KUKA KRL program: MyProgram_272().src

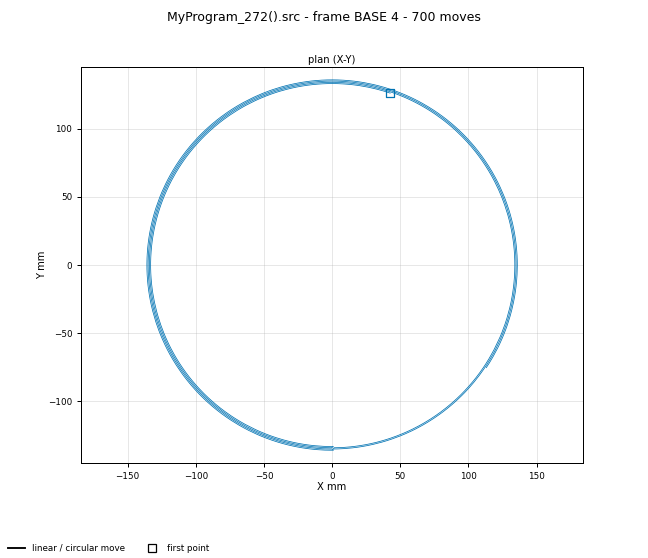
[picture p0: tool path of MyProgram_272().src in frame BASE 4, 700 of 700 moves have a stored position in this frame; points joined in program order, loops and branches not executed]
&ACCESS RVP
&REL 1
&PARAM TEMPLATE = C:\KRC\Roboter\Template\vorgabe
&PARAM EDITMASK = *
DEF MyProgram_272()
; ---- Setting reference (Base) ----
$BASE = BASE_DATA[4]

; --------------------------
; ---- Setting tool (TCP) ----
$TOOL = TOOL_DATA[3]
; --------------------------

$VEL.CP = VEL_APROX_PRINT
Startdeposition()
$VEL.CP = VEL_PRINT
LIN {X 42.5877,Y 126.1093,Z 171,A 71.929,B 9.2789,C 0.0558,E1 9.3306,E2 379.3226} C_DIS
LIN {X 38.192,Y 127.5107,Z 171,A 74.1551,B 9.2789,C 0.0493,E1 9.3246,E2 377.0683} C_DIS
LIN {X 32.5615,Y 129.0611,Z 171,A 76.4995,B 9.2789,C 0.0509,E1 9.3183,E2 374.7445} C_DIS
LIN {X 29.5199,Y 129.7905,Z 171,A 77.8234,B 9.2789,C 0.0505,E1 9.3147,E2 373.4236} C_DIS
LIN {X 26.303,Y 130.4807,Z 171,A 79.258,B 9.2789,C 0.0493,E1 9.3108,E2 371.9872} C_DIS
LIN {X 23.1123,Y 131.0837,Z 171,A 80.6058,B 9.2789,C 0.0496,E1 9.3071,E2 370.6457} C_DIS
LIN {X 20.0394,Y 131.5886,Z 171,A 81.9788,B 9.2789,C 0.0484,E1 9.3033,E2 369.2693} C_DIS
LIN {X 16.1157,Y 132.1266,Z 171,A 83.746,B 9.2789,C 0.0466,E1 9.2984,E2 367.4952} C_DIS
LIN {X 12.5078,Y 132.5166,Z 171,A 85.3108,B 9.2789,C 0.0461,E1 9.2941,E2 365.9307} C_DIS
LIN {X 8.3924,Y 132.8408,Z 171,A 87.0897,B 9.2789,C 0.0458,E1 9.2891,E2 364.1522} C_DIS
LIN {X 4.1202,Y 133.0424,Z 171,A 88.9439,B 9.2789,C 0.0454,E1 9.2839,E2 362.2973} C_DIS
LIN {X 0.5227,Y 133.1047,Z 171,A 90.4815,B 9.2789,C 0.0456,E1 9.2796,E2 360.7616} C_DIS
LIN {X -3.6809,Y 133.0546,Z 171,A 92.2437,B 9.2789,C 0.0466,E1 9.2747,E2 359.006} C_DIS
LIN {X -7.0154,Y 132.9209,Z 171,A 93.6521,B 9.2789,C 0.0474,E1 9.2708,E2 357.6017} C_DIS
LIN {X -10.707,Y 132.675,Z 171,A 95.3254,B 9.2789,C 0.0462,E1 9.2661,E2 355.9196} C_DIS
LIN {X -14.2828,Y 132.3368,Z 171,A 96.8212,B 9.2789,C 0.0477,E1 9.262,E2 354.4306} C_DIS
LIN {X -17.8991,Y 131.8978,Z 171,A 98.5277,B 9.2789,C 0.0457,E1 9.2572,E2 352.7086} C_DIS
LIN {X -21.9542,Y 131.2822,Z 171,A 100.1748,B 9.2789,C 0.0488,E1 9.2527,E2 351.0765} C_DIS
LIN {X -25.7118,Y 130.6003,Z 171,A 101.7895,B 9.2789,C 0.0503,E1 9.2483,E2 349.4665} C_DIS
LIN {X -29.321,Y 129.836,Z 171,A 103.4986,B 9.2789,C 0.049,E1 9.2436,E2 347.7439} C_DIS
LIN {X -33.1581,Y 128.9097,Z 171,A 105.1133,B 9.2789,C 0.0518,E1 9.2393,E2 346.1403} C_DIS
LIN {X -38.1705,Y 127.5171,Z 171,A 107.3466,B 9.2789,C 0.0538,E1 9.2333,E2 343.9094} C_DIS
LIN {X -40.8644,Y 126.6776,Z 171,A 108.5976,B 9.2789,C 0.0542,E1 9.2299,E2 342.6549} C_DIS
LIN {X -44.5339,Y 125.4356,Z 171,A 110.3593,B 9.2789,C 0.0542,E1 9.2253,E2 340.8833} C_DIS
LIN {X -48.093,Y 124.1129,Z 171,A 112.4224,B 9.2789,C 0.0481,E1 9.2198,E2 338.7703} C_DIS
LIN {X -52.2312,Y 122.4306,Z 171,A 113.7596,B 9.2789,C 0.0609,E1 9.2165,E2 337.5044} C_DIS
LIN {X -56.3646,Y 120.583,Z 171,A 115.8018,B 9.2789,C 0.0616,E1 9.2113,E2 335.4528} C_DIS
LIN {X -60.1833,Y 118.7221,Z 171,A 117.4022,B 9.2789,C 0.0681,E1 9.2073,E2 333.8809} C_DIS
LIN {X -62.74,Y 117.3935,Z 171,A 118.8099,B 9.2789,C 0.0669,E1 9.2038,E2 332.4544} C_DIS
LIN {X -65.4527,Y 115.9029,Z 171,A 120.3033,B 9.2789,C 0.0659,E1 9.2001,E2 330.9431} C_DIS
LIN {X -69.1961,Y 113.7079,Z 171,A 122.2249,B 9.2789,C 0.0678,E1 9.1955,E2 329.0167} C_DIS
LIN {X -73.1227,Y 111.2229,Z 171,A 123.9787,B 9.2788,C 0.0753,E1 9.1915,E2 327.2939} C_DIS
LIN {X -75.3901,Y 109.6986,Z 171,A 126.0091,B 9.2788,C 0.0623,E1 9.1866,E2 325.1627} C_DIS
LIN {X -79.6378,Y 106.655,Z 171,A 128.1469,B 9.2788,C 0.0683,E1 9.1818,E2 323.0405} C_DIS
LIN {X -83.2399,Y 103.8687,Z 171,A 129.6575,B 9.2788,C 0.0797,E1 9.1786,E2 321.5854} C_DIS
LIN {X -86.59,Y 101.0928,Z 171,A 131.612,B 9.2788,C 0.0818,E1 9.1744,E2 319.623} C_DIS
LIN {X -90.0311,Y 98.0401,Z 171,A 133.5166,B 9.2787,C 0.087,E1 9.1705,E2 317.7292} C_DIS
LIN {X -93.0134,Y 95.2157,Z 171,A 135.3296,B 9.2787,C 0.0899,E1 9.1669,E2 315.9127} C_DIS
LIN {X -95.7889,Y 92.4229,Z 171,A 137.1312,B 9.2787,C 0.0916,E1 9.1633,E2 314.1} C_DIS
LIN {X -99.0111,Y 88.9624,Z 171,A 139.1371,B 9.2786,C 0.0966,E1 9.1595,E2 312.0998} C_DIS
LIN {X -101.9431,Y 85.5866,Z 171,A 141.0403,B 9.2786,C 0.1012,E1 9.1561,E2 310.201} C_DIS
LIN {X -104.4924,Y 82.4553,Z 171,A 142.8577,B 9.2785,C 0.1039,E1 9.1529,E2 308.376} C_DIS
LIN {X -107.2539,Y 78.8293,Z 171,A 145.3979,B 9.2785,C 0.0988,E1 9.1486,E2 305.7684} C_DIS
LIN {X -110.2026,Y 74.6515,Z 171,A 147.0279,B 9.2784,C 0.1137,E1 9.1461,E2 304.2093} C_DIS
LIN {X -112.3849,Y 71.3246,Z 171,A 148.7665,B 9.2784,C 0.1175,E1 9.1435,E2 302.4694} C_DIS
LIN {X -114.8083,Y 67.3536,Z 171,A 150.9264,B 9.2784,C 0.1199,E1 9.1404,E2 300.2927} C_DIS
LIN {X -117.651,Y 62.2522,Z 171,A 153.1134,B 9.2781,C 0.1318,E1 9.1375,E2 298.1473} C_DIS
LIN {X -119.7398,Y 58.1376,Z 171,A 155.2917,B 9.2781,C 0.1338,E1 9.1347,E2 295.9483} C_DIS
LIN {X -121.0064,Y 55.4489,Z 171,A 156.578,B 9.2781,C 0.1371,E1 9.1332,E2 294.6624} C_DIS
LIN {X -122.3225,Y 52.4813,Z 171,A 158.0107,B 9.2781,C 0.1403,E1 9.1316,E2 293.227} C_DIS
LIN {X -123.8951,Y 48.6534,Z 171,A 159.9678,B 9.278,C 0.1422,E1 9.1296,E2 291.2507} C_DIS
LIN {X -125.2945,Y 44.9253,Z 171,A 161.607,B 9.278,C 0.1482,E1 9.128,E2 289.6223} C_DIS
LIN {X -126.5325,Y 41.3167,Z 171,A 163.3756,B 9.2779,C 0.1507,E1 9.1264,E2 287.8403} C_DIS
LIN {X -127.7786,Y 37.2777,Z 171,A 165.1311,B 9.2778,C 0.1568,E1 9.125,E2 286.0943} C_DIS
LIN {X -128.6977,Y 33.9703,Z 171,A 166.6461,B 9.2778,C 0.1604,E1 9.1239,E2 284.5764} C_DIS
LIN {X -129.8767,Y 29.1424,Z 171,A 168.7116,B 9.2776,C 0.1677,E1 9.1226,E2 282.5219} C_DIS
LIN {X -130.5951,Y 25.7359,Z 171,A 170.9382,B 9.2777,C 0.16,E1 9.1214,E2 280.2091} C_DIS
LIN {X -131.4748,Y 20.7743,Z 171,A 172.311,B 9.2774,C 0.1793,E1 9.1208,E2 278.9345} C_DIS
LIN {X -131.9531,Y 17.4769,Z 171,A 173.9819,B 9.2774,C 0.1796,E1 9.1201,E2 277.2366} C_DIS
LIN {X -132.405,Y 13.649,Z 171,A 175.7439,B 9.2773,C 0.1827,E1 9.1196,E2 275.4639} C_DIS
LIN {X -132.7511,Y 9.7054,Z 171,A 177.3737,B 9.2772,C 0.1889,E1 9.1192,E2 273.8447} C_DIS
LIN {X -132.9834,Y 5.7253,Z 171,A 179.185,B 9.2772,C 0.1923,E1 9.119,E2 272.0236} C_DIS
LIN {X -133.0886,Y 2.1253,Z 171,A -179.3539,B 9.277,C 0.1983,E1 9.1189,E2 270.5747} C_DIS
LIN {X -133.089,Y -2.0987,Z 171,A -177.4486,B 9.2769,C 0.2021,E1 9.1189,E2 268.6607} C_DIS
LIN {X -132.9791,Y -5.8335,Z 171,A -175.7236,B 9.2769,C 0.2049,E1 9.1191,E2 266.9232} C_DIS
LIN {X -132.7452,Y -9.7862,Z 171,A -174.0656,B 9.2767,C 0.2106,E1 9.1194,E2 265.2722} C_DIS
LIN {X -132.3555,Y -14.1094,Z 171,A -172.1851,B 9.2766,C 0.2158,E1 9.1199,E2 263.392} C_DIS
LIN {X -131.8984,Y -17.8939,Z 171,A -170.5736,B 9.2765,C 0.221,E1 9.1205,E2 261.7855} C_DIS
LIN {X -131.3884,Y -21.3181,Z 171,A -168.1542,B 9.2767,C 0.2099,E1 9.1217,E2 259.2544} C_DIS
LIN {X -130.2557,Y -27.4034,Z 171,A -166.3772,B 9.2762,C 0.2321,E1 9.1226,E2 257.5877} C_DIS
LIN {X -128.6414,Y -34.1817,Z 171,A -162.9035,B 9.2762,C 0.2327,E1 9.1249,E2 254.0589} C_DIS
LIN {X -127.6689,Y -37.652,Z 171,A -161.671,B 9.2759,C 0.2423,E1 9.1259,E2 252.8664} C_DIS
LIN {X -126.5371,Y -41.303,Z 171,A -160.0341,B 9.2759,C 0.2469,E1 9.1272,E2 251.2318} C_DIS
LIN {X -125.5991,Y -44.0688,Z 171,A -158.7983,B 9.2757,C 0.2507,E1 9.1284,E2 249.9995} C_DIS
LIN {X -124.5345,Y -46.9914,Z 171,A -157.3661,B 9.2757,C 0.2527,E1 9.1298,E2 248.557} C_DIS
LIN {X -123.3937,Y -49.9094,Z 171,A -155.9581,B 9.2756,C 0.2553,E1 9.1312,E2 247.1427} C_DIS
LIN {X -122.0333,Y -53.15,Z 171,A -154.4655,B 9.2755,C 0.2597,E1 9.1329,E2 245.6536} C_DIS
LIN {X -119.9685,Y -57.6591,Z 171,A -152.3072,B 9.2753,C 0.2648,E1 9.1354,E2 243.4938} C_DIS
LIN {X -118.1397,Y -61.3214,Z 171,A -150.483,B 9.2753,C 0.2682,E1 9.1377,E2 241.6632} C_DIS
LIN {X -115.8549,Y -65.5381,Z 171,A -148.4796,B 9.2751,C 0.2744,E1 9.1404,E2 239.6686} C_DIS
LIN {X -113.9926,Y -68.7254,Z 171,A -146.718,B 9.2751,C 0.2754,E1 9.143,E2 237.8869} C_DIS
LIN {X -111.7318,Y -72.3428,Z 171,A -144.854,B 9.2749,C 0.2793,E1 9.1458,E2 236.0204} C_DIS
LIN {X -109.9906,Y -74.9641,Z 171,A -143.532,B 9.2748,C 0.2831,E1 9.1478,E2 234.7031} C_DIS
LIN {X -107.4993,Y -78.4952,Z 171,A -141.6558,B 9.2747,C 0.2871,E1 9.1509,E2 232.8259} C_DIS
LIN {X -104.9019,Y -81.9339,Z 171,A -139.7691,B 9.2746,C 0.2907,E1 9.1541,E2 230.9362} C_DIS
LIN {X -102.8056,Y -84.5496,Z 171,A -138.2669,B 9.2745,C 0.2928,E1 9.1568,E2 229.4274} C_DIS
LIN {X -99.9648,Y -87.8898,Z 171,A -136.4848,B 9.2743,C 0.2987,E1 9.16,E2 227.6589} C_DIS
LIN {X -97.5072,Y -90.608,Z 171,A -134.6846,B 9.2743,C 0.298,E1 9.1634,E2 225.8321} C_DIS
LIN {X -94.0902,Y -94.1522,Z 171,A -132.586,B 9.2742,C 0.3026,E1 9.1676,E2 223.7367} C_DIS
LIN {X -90.8102,Y -97.3189,Z 171,A -130.6365,B 9.2741,C 0.3066,E1 9.1715,E2 221.7895} C_DIS
LIN {X -87.8913,Y -99.9635,Z 171,A -128.9777,B 9.2739,C 0.3104,E1 9.1749,E2 220.1357} C_DIS
LIN {X -84.6172,Y -102.7497,Z 171,A -127.0049,B 9.2739,C 0.3115,E1 9.1792,E2 218.1483} C_DIS
LIN {X -81.9414,Y -104.8961,Z 171,A -125.5632,B 9.2738,C 0.3147,E1 9.1824,E2 216.7112} C_DIS
LIN {X -78.4506,Y -107.5319,Z 171,A -123.6313,B 9.2738,C 0.3169,E1 9.1867,E2 214.7736} C_DIS
LIN {X -73.7879,Y -110.7828,Z 171,A -121.4632,B 9.2734,C 0.3257,E1 9.1916,E2 212.6402} C_DIS
LIN {X -71.2924,Y -112.4052,Z 171,A -119.8915,B 9.2735,C 0.3223,E1 9.1954,E2 211.0329} C_DIS
LIN {X -67.4694,Y -114.7403,Z 171,A -117.9853,B 9.2735,C 0.3254,E1 9.2,E2 209.1296} C_DIS
LIN {X -63.5644,Y -116.949,Z 171,A -115.9592,B 9.2734,C 0.3262,E1 9.2049,E2 207.0919} C_DIS
LIN {X -56.1378,Y -120.6878,Z 171,A -112.7264,B 9.273,C 0.3369,E1 9.2129,E2 203.9018} C_DIS
LIN {X -52.728,Y -122.2158,Z 171,A -110.8624,B 9.2731,C 0.3338,E1 9.2178,E2 202.0062} C_DIS
LIN {X -48.8795,Y -123.8072,Z 171,A -109.1519,B 9.2731,C 0.3371,E1 9.2222,E2 200.3059} C_DIS
LIN {X -45.6244,Y -125.0425,Z 171,A -107.7189,B 9.2729,C 0.3397,E1 9.2259,E2 198.8808} C_DIS
LIN {X -41.1313,Y -126.5923,Z 171,A -105.3843,B 9.273,C 0.3359,E1 9.2322,E2 196.5103} C_DIS
LIN {X -35.3399,Y -128.329,Z 171,A -102.9247,B 9.2729,C 0.3405,E1 9.2387,E2 194.0678} C_DIS
LIN {X -31.3297,Y -129.3656,Z 171,A -101.1229,B 9.2729,C 0.3411,E1 9.2436,E2 192.2633} C_DIS
LIN {X -28.0532,Y -130.1154,Z 171,A -99.6907,B 9.2729,C 0.3422,E1 9.2475,E2 190.8326} C_DIS
LIN {X -24.622,Y -130.8087,Z 171,A -98.045,B 9.2729,C 0.3401,E1 9.2521,E2 189.1693} C_DIS
LIN {X -20.5153,Y -131.5149,Z 171,A -96.3614,B 9.2728,C 0.3429,E1 9.2567,E2 187.4987} C_DIS
LIN {X -16.8361,Y -132.0371,Z 171,A -94.6911,B 9.2728,C 0.3419,E1 9.2613,E2 185.8191} C_DIS
LIN {X -12.5397,Y -132.5135,Z 171,A -92.9033,B 9.2728,C 0.3437,E1 9.2663,E2 184.0396} C_DIS
LIN {X -9.3135,Y -132.7797,Z 171,A -91.5471,B 9.2728,C 0.3446,E1 9.27,E2 182.6876} C_DIS
LIN {X -6.5086,Y -132.9463,Z 171,A -90.3022,B 9.2728,C 0.3439,E1 9.2735,E2 181.4378} C_DIS
LIN {X -2.5391,Y -133.0817,Z 171,A -88.4788,B 9.2728,C 0.3415,E1 9.2786,E2 179.5995} C_DIS
LIN {X 0.9624,Y -133.1014,Z 171,A -87.5259,B 9.2724,C 0.3524,E1 9.2811,E2 178.7143} C_DIS
Enddeposition()
LIN {X 0.9624,Y -133.1014,Z 171,A -87.5259,B 9.2724,C 0.3524,E1 9.2811,E2 178.7143} C_DIS
Startdeposition()
$VEL.CP = VEL_PRINT
LIN {X -0.4177,Y -134.0156,Z 171,A -88.5533,B 9.2717,C 0.3667,E1 9.2779,E2 179.8301} C_DIS
LIN {X -6.5028,Y -133.8581,Z 171,A -90.8877,B 9.272,C 0.3615,E1 9.2714,E2 182.1326} C_DIS
LIN {X -9.7045,Y -133.6639,Z 171,A -92.2371,B 9.272,C 0.3609,E1 9.2677,E2 183.4799} C_DIS
LIN {X -12.8663,Y -133.3967,Z 171,A -93.6193,B 9.272,C 0.3612,E1 9.2638,E2 184.8658} C_DIS
LIN {X -17.1502,Y -132.914,Z 171,A -95.4872,B 9.272,C 0.3613,E1 9.2586,E2 186.7374} C_DIS
LIN {X -20.4029,Y -132.4534,Z 171,A -96.8301,B 9.272,C 0.3597,E1 9.2549,E2 188.0732} C_DIS
LIN {X -23.3496,Y -131.9661,Z 171,A -98.1732,B 9.272,C 0.3605,E1 9.2512,E2 189.4248} C_DIS
LIN {X -26.8489,Y -131.2986,Z 171,A -99.7134,B 9.272,C 0.3602,E1 9.247,E2 190.9676} C_DIS
LIN {X -30.8258,Y -130.4234,Z 171,A -101.5112,B 9.272,C 0.3604,E1 9.2421,E2 192.7728} C_DIS
LIN {X -34.4158,Y -129.5211,Z 171,A -103.0201,B 9.272,C 0.358,E1 9.238,E2 194.273} C_DIS
LIN {X -38.4062,Y -128.3967,Z 171,A -105.2657,B 9.2718,C 0.3657,E1 9.2318,E2 196.577} C_DIS
LIN {X -42.1938,Y -127.2,Z 171,A -106.7736,B 9.272,C 0.3608,E1 9.2279,E2 198.0618} C_DIS
LIN {X -48.85,Y -124.7954,Z 171,A -109.5684,B 9.2722,C 0.3537,E1 9.2207,E2 200.8287} C_DIS
LIN {X -51.9025,Y -123.5569,Z 171,A -111.0717,B 9.2722,C 0.3541,E1 9.2167,E2 202.3436} C_DIS
LIN {X -55.8721,Y -121.8136,Z 171,A -112.7619,B 9.2724,C 0.3491,E1 9.2125,E2 204.0139} C_DIS
LIN {X -58.9006,Y -120.3785,Z 171,A -114.7479,B 9.2721,C 0.3576,E1 9.2073,E2 206.0676} C_DIS
LIN {X -62.6121,Y -118.4902,Z 171,A -116.1004,B 9.2725,C 0.3475,E1 9.2041,E2 207.3678} C_DIS
LIN {X -66.2758,Y -116.4825,Z 171,A -117.8773,B 9.2725,C 0.345,E1 9.1998,E2 209.1436} C_DIS
LIN {X -69.731,Y -114.4482,Z 171,A -119.4541,B 9.2727,C 0.3402,E1 9.196,E2 210.7034} C_DIS
LIN {X -72.5628,Y -112.6738,Z 171,A -121.1313,B 9.2727,C 0.3426,E1 9.192,E2 212.4109} C_DIS
LIN {X -75.4499,Y -110.7614,Z 171,A -122.4582,B 9.2728,C 0.3376,E1 9.189,E2 213.7188} C_DIS
LIN {X -80.2089,Y -107.3648,Z 171,A -125.1435,B 9.2728,C 0.3369,E1 9.1829,E2 216.4264} C_DIS
LIN {X -85.4194,Y -103.2673,Z 171,A -127.9742,B 9.273,C 0.3319,E1 9.1767,E2 219.2561} C_DIS
LIN {X -88.6446,Y -100.5126,Z 171,A -129.8183,B 9.2731,C 0.3292,E1 9.1728,E2 221.1034} C_DIS
LIN {X -92.9074,Y -96.5869,Z 171,A -132.4257,B 9.2732,C 0.3267,E1 9.1674,E2 223.726} C_DIS
LIN {X -96.4568,Y -93.0417,Z 171,A -134.2628,B 9.2736,C 0.3171,E1 9.1639,E2 225.5248} C_DIS
LIN {X -99.6208,Y -89.6461,Z 171,A -136.6709,B 9.2734,C 0.3204,E1 9.1593,E2 227.9838} C_DIS
LIN {X -103.0173,Y -85.7214,Z 171,A -138.7892,B 9.2737,C 0.3138,E1 9.1554,E2 230.0889} C_DIS
LIN {X -105.2838,Y -82.9215,Z 171,A -140.4396,B 9.2737,C 0.3123,E1 9.1526,E2 231.752} C_DIS
LIN {X -107.8412,Y -79.5674,Z 171,A -142.18,B 9.2739,C 0.3072,E1 9.1497,E2 233.484} C_DIS
LIN {X -110.346,Y -76.0555,Z 171,A -144.3303,B 9.2739,C 0.3081,E1 9.1462,E2 235.6704} C_DIS
LIN {X -112.4633,Y -72.8879,Z 171,A -145.6463,B 9.2742,C 0.2989,E1 9.1442,E2 236.9477} C_DIS
LIN {X -114.8314,Y -69.0974,Z 171,A -147.6104,B 9.2742,C 0.2952,E1 9.1413,E2 238.9171} C_DIS
LIN {X -116.912,Y -65.5151,Z 171,A -149.9633,B 9.2742,C 0.3005,E1 9.138,E2 241.339} C_DIS
LIN {X -119.2817,Y -61.0906,Z 171,A -151.4367,B 9.2746,C 0.2839,E1 9.1362,E2 242.7301} C_DIS
LIN {X -121.9044,Y -55.6758,Z 171,A -154.2197,B 9.2747,C 0.2808,E1 9.1329,E2 245.537} C_DIS
LIN {X -123.4427,Y -52.1759,Z 171,A -155.8103,B 9.2749,C 0.2757,E1 9.1311,E2 247.1211} C_DIS
LIN {X -124.879,Y -48.6347,Z 171,A -157.3022,B 9.2751,C 0.269,E1 9.1296,E2 248.5946} C_DIS
LIN {X -125.9626,Y -45.7562,Z 171,A -158.6353,B 9.2751,C 0.2658,E1 9.1283,E2 249.9291} C_DIS
LIN {X -127.0217,Y -42.7291,Z 171,A -159.9619,B 9.2753,C 0.2613,E1 9.1271,E2 251.2492} C_DIS
LIN {X -127.8099,Y -40.3112,Z 171,A -161.6774,B 9.2751,C 0.2687,E1 9.1256,E2 253.0396} C_DIS
LIN {X -128.9459,Y -36.5143,Z 171,A -162.9445,B 9.2754,C 0.257,E1 9.1246,E2 254.254} C_DIS
LIN {X -130.0995,Y -32.1694,Z 171,A -165.2419,B 9.2754,C 0.2578,E1 9.123,E2 256.5951} C_DIS
LIN {X -130.863,Y -28.9038,Z 171,A -166.2829,B 9.2757,C 0.2473,E1 9.1224,E2 257.5877} C_DIS
LIN {X -131.7429,Y -24.5771,Z 171,A -168.5727,B 9.2757,C 0.2485,E1 9.1212,E2 259.9242} C_DIS
LIN {X -132.3184,Y -21.2749,Z 171,A -169.779,B 9.2758,C 0.2408,E1 9.1206,E2 261.1022} C_DIS
LIN {X -132.8626,Y -17.5426,Z 171,A -171.4077,B 9.2759,C 0.2364,E1 9.12,E2 262.7313} C_DIS
LIN {X -133.33,Y -13.5609,Z 171,A -173.1482,B 9.2761,C 0.2319,E1 9.1195,E2 264.4735} C_DIS
LIN {X -133.6602,Y -9.7551,Z 171,A -174.78,B 9.2761,C 0.2271,E1 9.1191,E2 266.1037} C_DIS
LIN {X -133.8844,Y -5.98,Z 171,A -176.4973,B 9.2762,C 0.2241,E1 9.1188,E2 267.8317} C_DIS
LIN {X -133.9966,Y -2.2703,Z 171,A -178.0501,B 9.2764,C 0.2189,E1 9.1188,E2 269.3788} C_DIS
LIN {X -133.9984,Y 2.1614,Z 171,A -179.9463,B 9.2764,C 0.2135,E1 9.1188,E2 271.2734} C_DIS
LIN {X -133.8948,Y 5.7137,Z 171,A 178.3783,B 9.2765,C 0.2116,E1 9.1189,E2 272.9661} C_DIS
LIN {X -133.6354,Y 10.0951,Z 171,A 176.4685,B 9.2767,C 0.2067,E1 9.1193,E2 274.8779} C_DIS
LIN {X -133.254,Y 14.2681,Z 171,A 174.7796,B 9.2767,C 0.1998,E1 9.1198,E2 276.5528} C_DIS
LIN {X -132.8352,Y 17.7513,Z 171,A 173.1172,B 9.2768,C 0.1981,E1 9.1204,E2 278.2332} C_DIS
LIN {X -132.3596,Y 21.0091,Z 171,A 171.8075,B 9.277,C 0.1925,E1 9.1209,E2 279.5298} C_DIS
LIN {X -131.467,Y 26.0214,Z 171,A 169.4616,B 9.277,C 0.189,E1 9.1221,E2 281.8937} C_DIS
LIN {X -130.661,Y 29.7968,Z 171,A 167.9574,B 9.2772,C 0.1819,E1 9.123,E2 283.3787} C_DIS
LIN {X -129.8782,Y 33.0424,Z 171,A 166.4402,B 9.2772,C 0.1793,E1 9.124,E2 284.9052} C_DIS
LIN {X -128.9096,Y 36.6439,Z 171,A 164.8533,B 9.2773,C 0.1747,E1 9.1252,E2 286.4896} C_DIS
LIN {X -127.8259,Y 40.2612,Z 171,A 163.1507,B 9.2773,C 0.1716,E1 9.1266,E2 288.201} C_DIS
LIN {X -126.6485,Y 43.8211,Z 171,A 161.7514,B 9.2775,C 0.1638,E1 9.1278,E2 289.5744} C_DIS
LIN {X -124.6234,Y 49.2924,Z 171,A 158.8899,B 9.2775,C 0.163,E1 9.1307,E2 292.4771} C_DIS
LIN {X -123.083,Y 53.016,Z 171,A 157.2951,B 9.2776,C 0.1563,E1 9.1324,E2 294.0548} C_DIS
LIN {X -121.6103,Y 56.3119,Z 171,A 155.77,B 9.2777,C 0.1519,E1 9.1342,E2 295.5761} C_DIS
LIN {X -120.1754,Y 59.3123,Z 171,A 154.2867,B 9.2777,C 0.1491,E1 9.136,E2 297.0652} C_DIS
LIN {X -118.4959,Y 62.6012,Z 171,A 152.0812,B 9.2777,C 0.1553,E1 9.1389,E2 299.3431} C_DIS
LIN {X -116.1113,Y 66.9241,Z 171,A 150.7019,B 9.2779,C 0.1379,E1 9.1407,E2 300.6339} C_DIS
LIN {X -113.1851,Y 71.7622,Z 171,A 148.0619,B 9.2779,C 0.1356,E1 9.1446,E2 303.2979} C_DIS
LIN {X -110.5837,Y 75.7084,Z 171,A 145.5725,B 9.2779,C 0.1384,E1 9.1486,E2 305.8405} C_DIS
LIN {X -108.1591,Y 79.1347,Z 171,A 144.1073,B 9.278,C 0.1287,E1 9.1509,E2 307.2651} C_DIS
LIN {X -105.3435,Y 82.8454,Z 171,A 142.1606,B 9.2781,C 0.1233,E1 9.1542,E2 309.2045} C_DIS
LIN {X -103.2547,Y 85.4347,Z 171,A 140.6936,B 9.2781,C 0.1208,E1 9.1568,E2 310.6753} C_DIS
LIN {X -100.3672,Y 88.809,Z 171,A 138.7733,B 9.2782,C 0.1169,E1 9.1603,E2 312.5962} C_DIS
LIN {X -96.5571,Y 92.9381,Z 171,A 136.3014,B 9.2782,C 0.113,E1 9.1651,E2 315.074} C_DIS
LIN {X -93.2318,Y 96.2728,Z 171,A 134.3225,B 9.2783,C 0.1082,E1 9.169,E2 317.0469} C_DIS
LIN {X -90.1194,Y 99.1924,Z 171,A 132.7095,B 9.2783,C 0.1009,E1 9.1722,E2 318.633} C_DIS
LIN {X -87.0108,Y 101.9304,Z 171,A 130.6458,B 9.2783,C 0.1025,E1 9.1766,E2 320.7297} C_DIS
LIN {X -83.6922,Y 104.6724,Z 171,A 129.0731,B 9.2785,C 0.0945,E1 9.18,E2 322.269} C_DIS
LIN {X -80.3975,Y 107.2241,Z 171,A 126.6666,B 9.2784,C 0.1021,E1 9.1855,E2 324.7476} C_DIS
LIN {X -77.3007,Y 109.4769,Z 171,A 125.25,B 9.2784,C 0.0955,E1 9.1886,E2 326.1368} C_DIS
LIN {X -73.3191,Y 112.1833,Z 171,A 123.4063,B 9.2785,C 0.0884,E1 9.1929,E2 327.9533} C_DIS
LIN {X -69.7124,Y 114.4596,Z 171,A 121.3912,B 9.2785,C 0.0889,E1 9.1977,E2 329.9894} C_DIS
LIN {X -65.8282,Y 116.7361,Z 171,A 119.5565,B 9.2785,C 0.0844,E1 9.2021,E2 331.8118} C_DIS
LIN {X -61.9214,Y 118.8528,Z 171,A 117.1458,B 9.2785,C 0.0908,E1 9.2082,E2 334.281} C_DIS
LIN {X -58.0245,Y 120.8028,Z 171,A 115.7201,B 9.2785,C 0.0806,E1 9.2116,E2 335.6537} C_DIS
LIN {X -54.7944,Y 122.3016,Z 171,A 114.2618,B 9.2786,C 0.0776,E1 9.2153,E2 337.1032} C_DIS
LIN {X -52.003,Y 123.5149,Z 171,A 112.8217,B 9.2786,C 0.0786,E1 9.2191,E2 338.5587} C_DIS
LIN {X -44.0064,Y 126.5842,Z 171,A 109.2691,B 9.2786,C 0.0728,E1 9.2283,E2 342.0957} C_DIS
LIN {X -40.8891,Y 127.6253,Z 171,A 106.9838,B 9.2786,C 0.0874,E1 9.2347,E2 344.4831} C_DIS
LIN {X -34.9277,Y 129.3846,Z 171,A 105.1211,B 9.2786,C 0.0709,E1 9.2394,E2 346.2511} C_DIS
LIN {X -31.6163,Y 130.2329,Z 171,A 103.7268,B 9.2786,C 0.0686,E1 9.2432,E2 347.6365} C_DIS
LIN {X -28.2283,Y 131.0089,Z 171,A 102.2256,B 9.2786,C 0.0679,E1 9.2473,E2 349.1384} C_DIS
LIN {X -24.9215,Y 131.6782,Z 171,A 100.7058,B 9.2786,C 0.0685,E1 9.2515,E2 350.6665} C_DIS
LIN {X -21.097,Y 132.346,Z 171,A 99.0202,B 9.2786,C 0.0681,E1 9.2561,E2 352.3542} C_DIS
LIN {X -17.613,Y 132.8534,Z 171,A 97.5744,B 9.2786,C 0.0663,E1 9.2601,E2 353.7921} C_DIS
LIN {X -13.6517,Y 133.3203,Z 171,A 95.7637,B 9.2786,C 0.0678,E1 9.2651,E2 355.6143} C_DIS
LIN {X -9.871,Y 133.6518,Z 171,A 94.2447,B 9.2787,C 0.0654,E1 9.2693,E2 357.1202} C_DIS
LIN {X -6.1759,Y 133.8745,Z 171,A 92.591,B 9.2787,C 0.0664,E1 9.274,E2 358.7816} C_DIS
LIN {X -2.4995,Y 133.9928,Z 171,A 91.0689,B 9.2787,C 0.0653,E1 9.2782,E2 360.2969} C_DIS
LIN {X 1.5617,Y 134.0084,Z 171,A 89.2651,B 9.2787,C 0.0666,E1 9.2833,E2 362.1079} C_DIS
LIN {X 5.2476,Y 133.913,Z 171,A 87.7275,B 9.2787,C 0.0659,E1 9.2875,E2 363.6402} C_DIS
LIN {X 9.6343,Y 133.669,Z 171,A 85.9771,B 9.2787,C 0.0638,E1 9.2924,E2 365.3747} C_DIS
LIN {X 12.6886,Y 133.4137,Z 171,A 84.593,B 9.2787,C 0.0655,E1 9.2962,E2 366.767} C_DIS
LIN {X 16.5109,Y 132.9962,Z 171,A 82.9255,B 9.2787,C 0.0665,E1 9.3009,E2 368.4369} C_DIS
LIN {X 20.3126,Y 132.4674,Z 171,A 81.298,B 9.2787,C 0.0668,E1 9.3054,E2 370.0622} C_DIS
LIN {X 23.9999,Y 131.8497,Z 171,A 79.5993,B 9.2787,C 0.0696,E1 9.3101,E2 371.7723} C_DIS
LIN {X 27.9259,Y 131.0742,Z 171,A 77.9631,B 9.2787,C 0.0691,E1 9.3145,E2 373.3992} C_DIS
LIN {X 31.4693,Y 130.2683,Z 171,A 76.4813,B 9.2787,C 0.0686,E1 9.3185,E2 374.8722} C_DIS
LIN {X 34.5136,Y 129.495,Z 171,A 75.3185,B 9.2787,C 0.066,E1 9.3216,E2 376.0132} C_DIS
LIN {X 39.1117,Y 128.1812,Z 171,A 72.8281,B 9.2787,C 0.0765,E1 9.3284,E2 378.5562} C_DIS
LIN {X 42.5273,Y 127.0889,Z 171,A 71.232,B 9.2786,C 0.0792,E1 9.3327,E2 380.1596} C_DIS
LIN {X 45.9252,Y 125.9017,Z 171,A 70.0461,B 9.2786,C 0.0735,E1 9.3357,E2 381.3035} C_DIS
LIN {X 49.1641,Y 124.6732,Z 171,A 68.4441,B 9.2786,C 0.0775,E1 9.3399,E2 382.9198} C_DIS
LIN {X 52.9446,Y 123.1139,Z 171,A 66.8544,B 9.2786,C 0.0762,E1 9.3439,E2 384.4904} C_DIS
LIN {X 55.9136,Y 121.7945,Z 171,A 65.4645,B 9.2786,C 0.0778,E1 9.3475,E2 385.8804} C_DIS
LIN {X 59.0961,Y 120.2821,Z 171,A 64.0322,B 9.2786,C 0.0781,E1 9.351,E2 387.3039} C_DIS
LIN {X 62.0821,Y 118.7685,Z 171,A 62.6046,B 9.2786,C 0.0799,E1 9.3546,E2 388.7311} C_DIS
LIN {X 65.0999,Y 117.1438,Z 171,A 61.0728,B 9.2786,C 0.0833,E1 9.3584,E2 390.271} C_DIS
LIN {X 68.8077,Y 115.0051,Z 171,A 59.1857,B 9.2786,C 0.0871,E1 9.3629,E2 392.165} C_DIS
LIN {X 72.5733,Y 112.6671,Z 171,A 56.987,B 9.2784,C 0.0964,E1 9.3682,E2 394.4} C_DIS
LIN {X 75.7489,Y 110.5564,Z 171,A 55.3878,B 9.2784,C 0.0984,E1 9.3719,E2 395.9958} C_DIS
LIN {X 78.8374,Y 108.3759,Z 171,A 54.2058,B 9.2784,C 0.0919,E1 9.3744,E2 397.1264} C_DIS
LIN {X 81.2133,Y 106.6069,Z 171,A 52.7907,B 9.2784,C 0.0973,E1 9.3776,E2 398.5595} C_DIS
LIN {X 84.9683,Y 103.639,Z 171,A 50.8087,B 9.2784,C 0.0996,E1 9.3819,E2 400.5343} C_DIS
LIN {X 88.0703,Y 101.0161,Z 171,A 49.2958,B 9.2784,C 0.098,E1 9.3851,E2 402.0209} C_DIS
LIN {X 90.7394,Y 98.6254,Z 171,A 47.6034,B 9.2784,C 0.1044,E1 9.3886,E2 403.733} C_DIS
LIN {X 93.9387,Y 95.5832,Z 171,A 45.8588,B 9.2784,C 0.1051,E1 9.3921,E2 405.461} C_DIS
LIN {X 95.7522,Y 93.7664,Z 171,A 44.5586,B 9.2783,C 0.1117,E1 9.3947,E2 406.7859} C_DIS
LIN {X 98.9491,Y 90.3873,Z 171,A 42.6131,B 9.2783,C 0.1149,E1 9.3984,E2 408.727} C_DIS
LIN {X 101.8672,Y 87.0852,Z 171,A 40.94,B 9.2783,C 0.1144,E1 9.4014,E2 410.3756} C_DIS
LIN {X 105.162,Y 83.0752,Z 171,A 38.333,B 9.2781,C 0.1278,E1 9.4061,E2 413.0301} C_DIS
LIN {X 107.3697,Y 80.2023,Z 171,A 37.0612,B 9.2781,C 0.1254,E1 9.4082,E2 414.2694} C_DIS
LIN {X 109.9919,Y 76.5663,Z 171,A 35.1818,B 9.2781,C 0.129,E1 9.4112,E2 416.1453} C_DIS
LIN {X 112.52,Y 72.8005,Z 171,A 33.2961,B 9.278,C 0.1325,E1 9.4141,E2 418.0256} C_DIS
LIN {X 114.8247,Y 69.1085,Z 171,A 31.4015,B 9.278,C 0.1378,E1 9.4168,E2 419.9253} C_DIS
LIN {X 117.0367,Y 65.2933,Z 171,A 29.3977,B 9.2778,C 0.1452,E1 9.4196,E2 421.9445} C_DIS
LIN {X 119.2849,Y 61.0843,Z 171,A 27.7546,B 9.2778,C 0.1416,E1 9.4217,E2 423.5409} C_DIS
LIN {X 120.8415,Y 57.9435,Z 171,A 26.2444,B 9.2778,C 0.1457,E1 9.4236,E2 425.0536} C_DIS
LIN {X 122.1126,Y 55.2169,Z 171,A 24.8379,B 9.2778,C 0.1518,E1 9.4252,E2 426.4754} C_DIS
LIN {X 123.4991,Y 52.0408,Z 171,A 23.4751,B 9.2777,C 0.153,E1 9.4267,E2 427.8249} C_DIS
LIN {X 124.4698,Y 49.6748,Z 171,A 21.4671,B 9.2773,C 0.1763,E1 9.4289,E2 429.9434} C_DIS
LIN {X 126.7157,Y 43.6273,Z 171,A 20.0205,B 9.2777,C 0.1546,E1 9.4301,E2 431.2342} C_DIS
LIN {X 128.8322,Y 36.9188,Z 171,A 16.5791,B 9.2773,C 0.1727,E1 9.433,E2 434.731} C_DIS
LIN {X 129.8799,Y 33.0358,Z 171,A 15.0041,B 9.2773,C 0.1742,E1 9.4341,E2 436.2898} C_DIS
LIN {X 130.6382,Y 29.8969,Z 171,A 13.5962,B 9.2773,C 0.1787,E1 9.435,E2 437.7021} C_DIS
LIN {X 131.5103,Y 25.8,Z 171,A 11.809,B 9.2771,C 0.1837,E1 9.436,E2 439.4904} C_DIS
LIN {X 132.1803,Y 22.1032,Z 171,A 10.2832,B 9.2771,C 0.1865,E1 9.4367,E2 441.0077} C_DIS
LIN {X 132.7254,Y 18.5559,Z 171,A 8.728,B 9.277,C 0.1914,E1 9.4374,E2 442.5668} C_DIS
LIN {X 133.2232,Y 14.5547,Z 171,A 7.148,B 9.277,C 0.1931,E1 9.4379,E2 444.1308} C_DIS
LIN {X 133.5336,Y 11.3578,Z 171,A 5.7071,B 9.2768,C 0.1986,E1 9.4383,E2 445.5812} C_DIS
LIN {X 133.8035,Y 7.5697,Z 171,A 4.0121,B 9.2767,C 0.2049,E1 9.4386,E2 447.2865} C_DIS
LIN {X 133.9678,Y 3.5892,Z 171,A 2.4261,B 9.2767,C 0.2072,E1 9.4387,E2 448.8597} C_DIS
LIN {X 134.0178,Y -0.3225,Z 171,A 0.6529,B 9.2765,C 0.2143,E1 9.4387,E2 450.6469} C_DIS
LIN {X 133.9249,Y -4.9426,Z 171,A -0.9246,B 9.2765,C 0.211,E1 9.4387,E2 452.1775} C_DIS
LIN {X 133.7439,Y -8.5368,Z 171,A -2.7521,B 9.2763,C 0.2221,E1 9.4383,E2 454.0418} C_DIS
LIN {X 133.413,Y -12.6957,Z 171,A -4.4178,B 9.2763,C 0.2246,E1 9.4379,E2 455.6949} C_DIS
LIN {X 133.0146,Y -16.3565,Z 171,A -6.0549,B 9.2761,C 0.2306,E1 9.4374,E2 457.3413} C_DIS
LIN {X 132.4585,Y -20.3699,Z 171,A -7.6522,B 9.2761,C 0.2325,E1 9.4368,E2 458.9238} C_DIS
LIN {X 131.9284,Y -23.5599,Z 171,A -9.0526,B 9.2759,C 0.2369,E1 9.4361,E2 460.3277} C_DIS
LIN {X 131.2093,Y -27.2879,Z 171,A -10.6896,B 9.2759,C 0.2419,E1 9.4352,E2 461.9681} C_DIS
LIN {X 130.2531,Y -31.5325,Z 171,A -12.6285,B 9.2756,C 0.249,E1 9.434,E2 463.9185} C_DIS
LIN {X 128.2184,Y -38.9901,Z 171,A -15.7037,B 9.2756,C 0.2531,E1 9.4317,E2 466.9691} C_DIS
LIN {X 126.8211,Y -43.3232,Z 171,A -17.7242,B 9.2753,C 0.2602,E1 9.4299,E2 469.0007} C_DIS
LIN {X 125.5483,Y -46.8802,Z 171,A -19.1984,B 9.2753,C 0.2615,E1 9.4285,E2 470.4593} C_DIS
LIN {X 124.5217,Y -49.546,Z 171,A -20.5407,B 9.2751,C 0.2676,E1 9.4271,E2 471.8178} C_DIS
LIN {X 123.083,Y -53.016,Z 171,A -22.0256,B 9.2751,C 0.2692,E1 9.4255,E2 473.2895} C_DIS
LIN {X 118.707,Y -62.1992,Z 171,A -26.0129,B 9.275,C 0.2726,E1 9.4207,E2 477.237} C_DIS
LIN {X 115.054,Y -68.7257,Z 171,A -29.5125,B 9.2745,C 0.2877,E1 9.4159,E2 480.7775} C_DIS
LIN {X 112.6988,Y -72.5239,Z 171,A -31.4225,B 9.2744,C 0.2925,E1 9.413,E2 482.6894} C_DIS
LIN {X 110.7527,Y -75.4627,Z 171,A -33.2563,B 9.274,C 0.3035,E1 9.4101,E2 484.5649} C_DIS
LIN {X 108.43,Y -78.7627,Z 171,A -34.373,B 9.2743,C 0.2941,E1 9.4084,E2 485.6087} C_DIS
LIN {X 105.6597,Y -82.4428,Z 171,A -36.5823,B 9.274,C 0.3042,E1 9.4046,E2 487.8497} C_DIS
LIN {X 103.5506,Y -85.0765,Z 171,A -37.9109,B 9.274,C 0.305,E1 9.4022,E2 489.1658} C_DIS
LIN {X 100.3009,Y -88.884,Z 171,A -40.0893,B 9.2738,C 0.3107,E1 9.3983,E2 491.351} C_DIS
LIN {X 97.2492,Y -92.2135,Z 171,A -41.9997,B 9.2736,C 0.3145,E1 9.3946,E2 493.261} C_DIS
LIN {X 94.5132,Y -95.0151,Z 171,A -43.5453,B 9.2736,C 0.3153,E1 9.3916,E2 494.7924} C_DIS
LIN {X 91.0985,Y -98.2943,Z 171,A -45.663,B 9.2734,C 0.3215,E1 9.3873,E2 496.9237} C_DIS
LIN {X 87.832,Y -101.224,Z 171,A -47.5277,B 9.2733,C 0.3251,E1 9.3834,E2 498.7888} C_DIS
LIN {X 84.1009,Y -104.344,Z 171,A -50.2379,B 9.2727,C 0.3428,E1 9.3773,E2 501.5782} C_DIS
LIN {X 79.5271,Y -107.8708,Z 171,A -52.3896,B 9.2727,C 0.3404,E1 9.3726,E2 503.6935} C_DIS
LIN {X 76.0886,Y -110.3233,Z 171,A -53.7981,B 9.2729,C 0.335,E1 9.3695,E2 505.0549} C_DIS
LIN {X 72.5344,Y -112.692,Z 171,A -55.6305,B 9.2729,C 0.3382,E1 9.3652,E2 506.8898} C_DIS
LIN {X 67.5933,Y -115.7233,Z 171,A -58.5163,B 9.2724,C 0.3509,E1 9.3581,E2 509.8278} C_DIS
LIN {X 63.6006,Y -117.9645,Z 171,A -60.1009,B 9.2725,C 0.3459,E1 9.3544,E2 511.3683} C_DIS
LIN {X 58.7928,Y -120.4317,Z 171,A -62.3301,B 9.2725,C 0.3474,E1 9.3488,E2 513.5895} C_DIS
LIN {X 55.1887,Y -122.1252,Z 171,A -63.9376,B 9.2725,C 0.3477,E1 9.3448,E2 515.1866} C_DIS
LIN {X 51.9283,Y -123.5461,Z 171,A -65.4403,B 9.2725,C 0.3492,E1 9.3409,E2 516.6883} C_DIS
LIN {X 47.5193,Y -125.3089,Z 171,A -67.654,B 9.2722,C 0.3554,E1 9.3351,E2 518.9264} C_DIS
LIN {X 42.6137,Y -127.0601,Z 171,A -69.6647,B 9.2722,C 0.3533,E1 9.3298,E2 520.912} C_DIS
LIN {X 39.2717,Y -128.1322,Z 171,A -71.1302,B 9.2722,C 0.354,E1 9.3259,E2 522.3743} C_DIS
LIN {X 35.5623,Y -129.2121,Z 171,A -72.8911,B 9.2721,C 0.3578,E1 9.3212,E2 524.1499} C_DIS
LIN {X 31.9286,Y -130.1576,Z 171,A -74.4546,B 9.2721,C 0.3583,E1 9.3169,E2 525.7094} C_DIS
LIN {X 28.2761,Y -130.9986,Z 171,A -75.9609,B 9.2721,C 0.3575,E1 9.3129,E2 527.2048} C_DIS
LIN {X 24.7618,Y -131.7087,Z 171,A -77.5544,B 9.2721,C 0.3598,E1 9.3085,E2 528.8069} C_DIS
LIN {X 20.5857,Y -132.4251,Z 171,A -79.3414,B 9.272,C 0.3603,E1 9.3036,E2 530.5919} C_DIS
LIN {X 16.4998,Y -132.9975,Z 171,A -81.1056,B 9.272,C 0.3613,E1 9.2987,E2 532.3573} C_DIS
LIN {X 13.314,Y -133.3537,Z 171,A -82.5894,B 9.2718,C 0.3641,E1 9.2945,E2 533.8558} C_DIS
LIN {X 8.8975,Y -133.7217,Z 171,A -84.6293,B 9.2718,C 0.3677,E1 9.2888,E2 535.9147} C_DIS
LIN {X 5.628,Y -133.8982,Z 171,A -85.8371,B 9.2718,C 0.3642,E1 9.2855,E2 537.0996} C_DIS
LIN {X 1.4185,Y -134.01,Z 171,A -87.5737,B 9.2718,C 0.3632,E1 9.2806,E2 538.8292} C_DIS
LIN {X 1.4185,Y -134.01,Z 171,A -87.5737,B 9.2718,C 0.3632,E1 9.2806,E2 538.8292} C_DIS
Enddeposition()
LIN {X 0.9732,Y -134.9202,Z 171,A -87.2182,B 9.1317,C 0.3614,E1 9.1414,E2 538.4809} C_DIS
Startdeposition()
$VEL.CP = VEL_PRINT
LIN {X 3.8946,Y -134.87,Z 171,A -85.157,B 9.1323,C 0.3446,E1 9.1475,E2 536.3156} C_DIS
LIN {X 8.7184,Y -134.6448,Z 171,A -83.8575,B 9.1318,C 0.3592,E1 9.1509,E2 535.1102} C_DIS
LIN {X 12.2227,Y -134.372,Z 171,A -82.3078,B 9.1318,C 0.3575,E1 9.1552,E2 533.5524} C_DIS
LIN {X 14.9924,Y -134.0916,Z 171,A -80.9558,B 9.132,C 0.3536,E1 9.159,E2 532.1784} C_DIS
LIN {X 18.9403,Y -133.59,Z 171,A -79.3608,B 9.132,C 0.3546,E1 9.1634,E2 530.5943} C_DIS
LIN {X 22.2327,Y -133.0816,Z 171,A -77.912,B 9.132,C 0.3531,E1 9.1674,E2 529.1403} C_DIS
LIN {X 26.0347,Y -132.3922,Z 171,A -76.1666,B 9.1321,C 0.3499,E1 9.1722,E2 527.3807} C_DIS
LIN {X 30.0092,Y -131.5463,Z 171,A -74.5867,B 9.1321,C 0.3516,E1 9.1765,E2 525.8181} C_DIS
LIN {X 33.4879,Y -130.7043,Z 171,A -73.1084,B 9.1321,C 0.3512,E1 9.1805,E2 524.3439} C_DIS
LIN {X 36.5496,Y -129.8812,Z 171,A -71.7043,B 9.1321,C 0.3488,E1 9.1843,E2 522.9316} C_DIS
LIN {X 39.7422,Y -128.9402,Z 171,A -70.2431,B 9.1323,C 0.3465,E1 9.1882,E2 521.4633} C_DIS
LIN {X 43.7664,Y -127.6309,Z 171,A -68.4844,B 9.1323,C 0.3454,E1 9.1928,E2 519.7081} C_DIS
LIN {X 49.8363,Y -125.3862,Z 171,A -65.8719,B 9.1323,C 0.3452,E1 9.1997,E2 517.1107} C_DIS
LIN {X 53.8643,Y -123.708,Z 171,A -63.8778,B 9.1325,C 0.3398,E1 9.2048,E2 515.0973} C_DIS
LIN {X 58.3399,Y -121.661,Z 171,A -61.8664,B 9.1325,C 0.3387,E1 9.2099,E2 513.0941} C_DIS
LIN {X 61.3653,Y -120.1633,Z 171,A -60.4716,B 9.1325,C 0.3375,E1 9.2134,E2 511.7029} C_DIS
LIN {X 65.8598,Y -117.7619,Z 171,A -58.091,B 9.1329,C 0.3296,E1 9.2193,E2 509.2932} C_DIS
LIN {X 70.2272,Y -115.2117,Z 171,A -56.3609,B 9.1327,C 0.3353,E1 9.2233,E2 507.6139} C_DIS
LIN {X 74.4482,Y -112.53,Z 171,A -53.9842,B 9.133,C 0.3262,E1 9.229,E2 505.2033} C_DIS
LIN {X 78.7278,Y -109.5786,Z 171,A -52.0507,B 9.133,C 0.3283,E1 9.2333,E2 503.3024} C_DIS
LIN {X 81.1914,Y -107.7655,Z 171,A -50.1645,B 9.1335,C 0.3131,E1 9.2377,E2 501.3407} C_DIS
LIN {X 84.4433,Y -105.2373,Z 171,A -48.789,B 9.1333,C 0.318,E1 9.2406,E2 500.0109} C_DIS
LIN {X 87.8145,Y -102.441,Z 171,A -46.9109,B 9.1334,C 0.3139,E1 9.2446,E2 498.1287} C_DIS
LIN {X 91.2042,Y -99.4347,Z 171,A -45.0502,B 9.1335,C 0.3114,E1 9.2484,E2 496.274} C_DIS
LIN {X 95.0316,Y -95.7834,Z 171,A -43.008,B 9.1335,C 0.3112,E1 9.2525,E2 494.2554} C_DIS
LIN {X 97.4118,Y -93.3618,Z 171,A -41.399,B 9.1337,C 0.3044,E1 9.2557,E2 492.6239} C_DIS
LIN {X 100.3412,Y -90.2062,Z 171,A -39.5702,B 9.1339,C 0.3003,E1 9.2591,E2 490.7931} C_DIS
LIN {X 104.0484,Y -85.9035,Z 171,A -37.4453,B 9.1339,C 0.3013,E1 9.2629,E2 488.7019} C_DIS
LIN {X 106.0595,Y -83.4076,Z 171,A -35.6831,B 9.1342,C 0.2891,E1 9.2661,E2 486.8878} C_DIS
LIN {X 108.0256,Y -80.8457,Z 171,A -34.6365,B 9.1342,C 0.2931,E1 9.2677,E2 485.8807} C_DIS
LIN {X 111.1695,Y -76.4645,Z 171,A -32.2758,B 9.1343,C 0.2859,E1 9.2716,E2 483.5088} C_DIS
LIN {X 113.5673,Y -72.8555,Z 171,A -30.4338,B 9.1345,C 0.2813,E1 9.2744,E2 481.6645} C_DIS
LIN {X 115.8862,Y -69.1074,Z 171,A -28.0764,B 9.135,C 0.2655,E1 9.2779,E2 479.2438} C_DIS
LIN {X 118.3687,Y -64.7638,Z 171,A -26.7717,B 9.1346,C 0.2787,E1 9.2795,E2 478.0403} C_DIS
LIN {X 119.8092,Y -62.0583,Z 171,A -25.1718,B 9.1349,C 0.2685,E1 9.2816,E2 476.4016} C_DIS
LIN {X 123.5957,Y -54.124,Z 171,A -21.7143,B 9.1349,C 0.2648,E1 9.2857,E2 472.975} C_DIS
LIN {X 124.5582,Y -51.867,Z 171,A -20.6097,B 9.1351,C 0.2605,E1 9.2869,E2 471.8613} C_DIS
LIN {X 125.8734,Y -48.5892,Z 171,A -19.1102,B 9.1352,C 0.2564,E1 9.2884,E2 470.3603} C_DIS
LIN {X 127.577,Y -43.9218,Z 171,A -17.063,B 9.1353,C 0.252,E1 9.2903,E2 468.3188} C_DIS
LIN {X 128.6291,Y -40.7382,Z 171,A -15.6551,B 9.1354,C 0.2484,E1 9.2915,E2 466.9114} C_DIS
LIN {X 129.6608,Y -37.3282,Z 171,A -13.3482,B 9.136,C 0.2259,E1 9.2934,E2 464.503} C_DIS
LIN {X 131.195,Y -31.5095,Z 171,A -11.6275,B 9.1357,C 0.2379,E1 9.2945,E2 462.8848} C_DIS
LIN {X 132.0315,Y -27.8055,Z 171,A -9.9853,B 9.1358,C 0.2326,E1 9.2955,E2 461.2373} C_DIS
LIN {X 132.8067,Y -23.8197,Z 171,A -8.3507,B 9.1359,C 0.2297,E1 9.2963,E2 459.6121} C_DIS
LIN {X 133.3897,Y -20.3056,Z 171,A -6.7921,B 9.136,C 0.2242,E1 9.297,E2 458.0463} C_DIS
LIN {X 133.9595,Y -16.1214,Z 171,A -5.1089,B 9.1361,C 0.2216,E1 9.2976,E2 456.375} C_DIS
LIN {X 134.3129,Y -12.8481,Z 171,A -3.7121,B 9.1362,C 0.2175,E1 9.298,E2 454.977} C_DIS
LIN {X 134.6427,Y -8.7516,Z 171,A -1.8421,B 9.1364,C 0.2096,E1 9.2983,E2 453.0898} C_DIS
LIN {X 134.8394,Y -4.854,Z 171,A -0.4293,B 9.1364,C 0.2104,E1 9.2985,E2 451.7059} C_DIS
LIN {X 134.9199,Y -1.4957,Z 171,A 1.0951,B 9.1365,C 0.204,E1 9.2985,E2 450.1679} C_DIS
LIN {X 134.9026,Y 2.5398,Z 171,A 2.7369,B 9.1365,C 0.2007,E1 9.2985,E2 448.5334} C_DIS
LIN {X 134.7612,Y 6.6695,Z 171,A 4.473,B 9.1367,C 0.196,E1 9.2983,E2 446.7981} C_DIS
LIN {X 134.529,Y 10.3579,Z 171,A 6.0024,B 9.1367,C 0.1924,E1 9.298,E2 445.2722} C_DIS
LIN {X 134.1608,Y 14.3497,Z 171,A 7.6722,B 9.1369,C 0.1882,E1 9.2976,E2 443.6049} C_DIS
LIN {X 133.7629,Y 17.678,Z 171,A 9.03,B 9.1369,C 0.1856,E1 9.2971,E2 442.254} C_DIS
LIN {X 133.2617,Y 21.1321,Z 171,A 10.5071,B 9.1369,C 0.1815,E1 9.2965,E2 440.7762} C_DIS
LIN {X 132.5741,Y 25.0832,Z 171,A 12.2121,B 9.1371,C 0.1766,E1 9.2956,E2 439.0696} C_DIS
LIN {X 131.8711,Y 28.5484,Z 171,A 13.6313,B 9.1371,C 0.1742,E1 9.2948,E2 437.6593} C_DIS
LIN {X 131.1534,Y 31.6823,Z 171,A 15.0052,B 9.1372,C 0.1701,E1 9.2939,E2 436.2832} C_DIS
LIN {X 130.2816,Y 35.0969,Z 171,A 16.5203,B 9.1372,C 0.1655,E1 9.2929,E2 434.7647} C_DIS
LIN {X 128.3507,Y 41.61,Z 171,A 19.3012,B 9.1374,C 0.1599,E1 9.2906,E2 431.9945} C_DIS
LIN {X 127.2235,Y 44.9414,Z 171,A 20.7781,B 9.1374,C 0.1562,E1 9.2893,E2 430.5186} C_DIS
LIN {X 125.3326,Y 49.9692,Z 171,A 22.9192,B 9.1375,C 0.1532,E1 9.2872,E2 428.3931} C_DIS
LIN {X 123.7314,Y 53.8102,Z 171,A 24.8035,B 9.1376,C 0.1459,E1 9.2851,E2 426.4932} C_DIS
LIN {X 122.4187,Y 56.7326,Z 171,A 26.1836,B 9.1376,C 0.1419,E1 9.2835,E2 425.1097} C_DIS
LIN {X 120.841,Y 60.0207,Z 171,A 27.6417,B 9.1377,C 0.1399,E1 9.2817,E2 423.6618} C_DIS
LIN {X 119.2505,Y 63.1223,Z 171,A 29.1763,B 9.1377,C 0.1349,E1 9.2797,E2 422.1196} C_DIS
LIN {X 117.194,Y 66.8657,Z 171,A 30.7914,B 9.1377,C 0.1348,E1 9.2775,E2 420.5279} C_DIS
LIN {X 115.4121,Y 69.8963,Z 171,A 32.356,B 9.1379,C 0.1295,E1 9.2753,E2 418.9537} C_DIS
LIN {X 113.387,Y 73.1368,Z 171,A 34.0651,B 9.1379,C 0.1237,E1 9.2727,E2 417.2331} C_DIS
LIN {X 111.0807,Y 76.5938,Z 171,A 35.8328,B 9.138,C 0.1194,E1 9.2699,E2 415.4642} C_DIS
LIN {X 108.5063,Y 80.1997,Z 171,A 37.6985,B 9.138,C 0.1154,E1 9.2669,E2 413.5994} C_DIS
LIN {X 104.0469,Y 85.9053,Z 171,A 40.4461,B 9.138,C 0.1157,E1 9.2622,E2 410.8907} C_DIS
LIN {X 101.9752,Y 88.3554,Z 171,A 42.0505,B 9.1381,C 0.1074,E1 9.2592,E2 409.2562} C_DIS
LIN {X 99.0004,Y 91.6761,Z 171,A 43.9294,B 9.1381,C 0.1037,E1 9.2557,E2 407.3784} C_DIS
LIN {X 95.7177,Y 95.0977,Z 171,A 45.9045,B 9.1382,C 0.1004,E1 9.2518,E2 405.4072} C_DIS
LIN {X 92.5831,Y 98.152,Z 171,A 47.7341,B 9.1382,C 0.0973,E1 9.2481,E2 403.5805} C_DIS
LIN {X 89.017,Y 101.3981,Z 171,A 49.6662,B 9.1382,C 0.0959,E1 9.2442,E2 401.662} C_DIS
LIN {X 85.6553,Y 104.2533,Z 171,A 51.6509,B 9.1383,C 0.0901,E1 9.2399,E2 399.6632} C_DIS
LIN {X 81.6561,Y 107.4145,Z 171,A 53.7812,B 9.1383,C 0.087,E1 9.2352,E2 397.5367} C_DIS
LIN {X 78.0746,Y 110.0452,Z 171,A 56.131,B 9.1385,C 0.074,E1 9.2297,E2 395.1298} C_DIS
LIN {X 74.1314,Y 112.7386,Z 171,A 57.5821,B 9.1385,C 0.0831,E1 9.2265,E2 393.749} C_DIS
LIN {X 70.7649,Y 114.8819,Z 171,A 59.3633,B 9.1385,C 0.0787,E1 9.2223,E2 391.9571} C_DIS
LIN {X 67.586,Y 116.7801,Z 171,A 60.7306,B 9.1385,C 0.0807,E1 9.219,E2 390.6147} C_DIS
LIN {X 64.2654,Y 118.6405,Z 171,A 62.51,B 9.1385,C 0.0751,E1 9.2146,E2 388.8154} C_DIS
LIN {X 60.9284,Y 120.3858,Z 171,A 63.9867,B 9.1385,C 0.0755,E1 9.211,E2 387.3535} C_DIS
LIN {X 57.8388,Y 121.9004,Z 171,A 65.4595,B 9.1385,C 0.0735,E1 9.2073,E2 385.8793} C_DIS
LIN {X 54.7574,Y 123.3153,Z 171,A 66.8884,B 9.1385,C 0.072,E1 9.2037,E2 384.4517} C_DIS
LIN {X 50.827,Y 124.9868,Z 171,A 68.6902,B 9.1385,C 0.0703,E1 9.199,E2 382.6515} C_DIS
LIN {X 47.6929,Y 126.216,Z 171,A 70.2769,B 9.1385,C 0.0656,E1 9.1948,E2 381.0458} C_DIS
LIN {X 43.6161,Y 127.683,Z 171,A 72.0376,B 9.1385,C 0.0656,E1 9.1902,E2 379.295} C_DIS
LIN {X 36.4175,Y 129.9182,Z 171,A 75.1311,B 9.1385,C 0.0651,E1 9.182,E2 376.2152} C_DIS
LIN {X 32.938,Y 130.8439,Z 171,A 76.6026,B 9.1385,C 0.0651,E1 9.178,E2 374.7509} C_DIS
LIN {X 29.7417,Y 131.6074,Z 171,A 78.031,B 9.1385,C 0.0636,E1 9.1741,E2 373.3189} C_DIS
LIN {X 25.7339,Y 132.4497,Z 171,A 79.7862,B 9.1385,C 0.0624,E1 9.1693,E2 371.5623} C_DIS
LIN {X 22.2868,Y 133.0726,Z 171,A 81.2729,B 9.1385,C 0.0617,E1 9.1652,E2 370.0761} C_DIS
LIN {X 18.9503,Y 133.5886,Z 171,A 82.709,B 9.1385,C 0.0611,E1 9.1613,E2 368.6402} C_DIS
LIN {X 14.8623,Y 134.1056,Z 171,A 84.4915,B 9.1385,C 0.0599,E1 9.1563,E2 366.8543} C_DIS
LIN {X 11.1463,Y 134.465,Z 171,A 86.0256,B 9.1385,C 0.0605,E1 9.1521,E2 365.3269} C_DIS
LIN {X 6.9263,Y 134.7483,Z 171,A 87.8059,B 9.1385,C 0.0605,E1 9.1471,E2 363.5493} C_DIS
LIN {X 3.5428,Y 134.8798,Z 171,A 89.2523,B 9.1385,C 0.0603,E1 9.1431,E2 362.1025} C_DIS
LIN {X -0.6476,Y 134.9246,Z 171,A 91.0369,B 9.1385,C 0.0602,E1 9.1381,E2 360.318} C_DIS
LIN {X -4.4004,Y 134.8559,Z 171,A 92.7188,B 9.1385,C 0.0587,E1 9.1334,E2 358.6263} C_DIS
LIN {X -8.2579,Y 134.6731,Z 171,A 94.27,B 9.1385,C 0.0607,E1 9.1291,E2 357.0867} C_DIS
LIN {X -12.1148,Y 134.3832,Z 171,A 96.0439,B 9.1385,C 0.0586,E1 9.1241,E2 355.2978} C_DIS
LIN {X -16.0199,Y 133.9716,Z 171,A 97.5738,B 9.1385,C 0.0618,E1 9.1199,E2 353.7854} C_DIS
LIN {X -19.4928,Y 133.5111,Z 171,A 99.0623,B 9.1385,C 0.0624,E1 9.1158,E2 352.2977} C_DIS
LIN {X -23.6069,Y 132.8448,Z 171,A 100.8611,B 9.1385,C 0.0628,E1 9.1108,E2 350.4964} C_DIS
LIN {X -27.292,Y 132.1374,Z 171,A 102.5455,B 9.1385,C 0.062,E1 9.1062,E2 348.8021} C_DIS
LIN {X -31.5919,Y 131.1752,Z 171,A 104.3038,B 9.1385,C 0.0654,E1 9.1014,E2 347.0586} C_DIS
LIN {X -34.7642,Y 130.3703,Z 171,A 106.5462,B 9.1386,C 0.0507,E1 9.0951,E2 344.7135} C_DIS
LIN {X -40.6516,Y 128.6568,Z 171,A 108.1638,B 9.1386,C 0.0711,E1 9.0911,E2 343.2176} C_DIS
LIN {X -43.424,Y 127.7496,Z 171,A 110.7264,B 9.1386,C 0.048,E1 9.084,E2 340.4949} C_DIS
LIN {X -50.6283,Y 125.0669,Z 171,A 112.8818,B 9.1385,C 0.0719,E1 9.0787,E2 338.4774} C_DIS
LIN {X -53.9549,Y 123.6688,Z 171,A 114.3908,B 9.1385,C 0.0741,E1 9.0748,E2 336.9724} C_DIS
LIN {X -57.405,Y 122.1077,Z 171,A 116.4463,B 9.1385,C 0.0681,E1 9.0695,E2 334.8641} C_DIS
LIN {X -60.8303,Y 120.4357,Z 171,A 117.8992,B 9.1385,C 0.0732,E1 9.0659,E2 333.4325} C_DIS
LIN {X -64.8994,Y 118.2947,Z 171,A 119.7284,B 9.1385,C 0.0781,E1 9.0615,E2 331.62} C_DIS
LIN {X -69.1683,Y 115.8499,Z 171,A 121.7278,B 9.1385,C 0.0828,E1 9.0567,E2 329.6332} C_DIS
LIN {X -72.0311,Y 114.0919,Z 171,A 123.2515,B 9.1384,C 0.0833,E1 9.053,E2 328.099} C_DIS
LIN {X -75.8499,Y 111.5899,Z 171,A 125.5741,B 9.1384,C 0.0798,E1 9.0475,E2 325.7317} C_DIS
LIN {X -79.1683,Y 109.2601,Z 171,A 126.999,B 9.1384,C 0.0879,E1 9.0444,E2 324.3444} C_DIS
LIN {X -82.901,Y 106.4564,Z 171,A 128.7699,B 9.1383,C 0.0952,E1 9.0405,E2 322.6009} C_DIS
LIN {X -85.5872,Y 104.3089,Z 171,A 130.4222,B 9.1383,C 0.0946,E1 9.0369,E2 320.9268} C_DIS
LIN {X -89.5415,Y 100.9344,Z 171,A 132.6456,B 9.1383,C 0.0985,E1 9.0322,E2 318.7036} C_DIS
LIN {X -91.7901,Y 98.8942,Z 171,A 133.9898,B 9.1383,C 0.1002,E1 9.0294,E2 317.354} C_DIS
LIN {X -94.4492,Y 96.3577,Z 171,A 135.3622,B 9.1382,C 0.1066,E1 9.0267,E2 316.0059} C_DIS
LIN {X -97.0032,Y 93.7861,Z 171,A 137.1765,B 9.1382,C 0.1051,E1 9.0231,E2 314.1598} C_DIS
LIN {X -100.2611,Y 90.2956,Z 171,A 139.0302,B 9.1381,C 0.1125,E1 9.0197,E2 312.3292} C_DIS
LIN {X -102.686,Y 87.5275,Z 171,A 140.5782,B 9.1381,C 0.1162,E1 9.0168,E2 310.7844} C_DIS
LIN {X -104.9835,Y 84.758,Z 171,A 142.2929,B 9.1381,C 0.1165,E1 9.0138,E2 309.0487} C_DIS
LIN {X -107.6787,Y 81.3064,Z 171,A 144.1615,B 9.138,C 0.1207,E1 9.0106,E2 307.181} C_DIS
LIN {X -111.7446,Y 75.6214,Z 171,A 147.081,B 9.1379,C 0.1286,E1 9.0059,E2 304.2705} C_DIS
LIN {X -113.9216,Y 72.3009,Z 171,A 148.9036,B 9.1379,C 0.1305,E1 9.0031,E2 302.4331} C_DIS
LIN {X -116.1896,Y 68.5968,Z 171,A 150.7192,B 9.1378,C 0.1356,E1 9.0005,E2 300.6229} C_DIS
LIN {X -119.3408,Y 62.9502,Z 171,A 153.22,B 9.1376,C 0.1467,E1 8.9972,E2 298.1546} C_DIS
LIN {X -121.1114,Y 59.4727,Z 171,A 155.1372,B 9.1376,C 0.1467,E1 8.9948,E2 296.2077} C_DIS
LIN {X -122.582,Y 56.3795,Z 171,A 156.5831,B 9.1376,C 0.1508,E1 8.993,E2 294.7643} C_DIS
LIN {X -124.0047,Y 53.1782,Z 171,A 158.0834,B 9.1375,C 0.1546,E1 8.9914,E2 293.2641} C_DIS
LIN {X -125.3768,Y 49.8596,Z 171,A 159.9233,B 9.1375,C 0.1535,E1 8.9894,E2 291.3874} C_DIS
LIN {X -127.7532,Y 43.4137,Z 171,A 162.6221,B 9.1373,C 0.1651,E1 8.9869,E2 288.7183} C_DIS
LIN {X -128.5927,Y 40.8522,Z 171,A 163.7882,B 9.1373,C 0.168,E1 8.9859,E2 287.5508} C_DIS
LIN {X -129.6014,Y 37.5312,Z 171,A 165.3299,B 9.1372,C 0.171,E1 8.9847,E2 286.0023} C_DIS
LIN {X -130.5391,Y 34.1312,Z 171,A 166.961,B 9.1372,C 0.173,E1 8.9835,E2 284.3565} C_DIS
LIN {X -131.5395,Y 30.0391,Z 171,A 168.6358,B 9.137,C 0.18,E1 8.9824,E2 282.6974} C_DIS
LIN {X -132.3185,Y 26.4022,Z 171,A 170.225,B 9.137,C 0.1843,E1 8.9815,E2 281.1086} C_DIS
LIN {X -133.2444,Y 21.244,Z 171,A 172.4045,B 9.1368,C 0.1915,E1 8.9805,E2 278.937} C_DIS
LIN {X -133.7559,Y 17.7319,Z 171,A 174.0505,B 9.1368,C 0.1935,E1 8.9798,E2 277.2756} C_DIS
LIN {X -134.1797,Y 14.174,Z 171,A 175.5883,B 9.1367,C 0.1977,E1 8.9794,E2 275.7373} C_DIS
LIN {X -134.5555,Y 9.9946,Z 171,A 177.4313,B 9.1366,C 0.2019,E1 8.9789,E2 273.8885} C_DIS
LIN {X -134.7593,Y 6.7075,Z 171,A 178.7937,B 9.1365,C 0.2065,E1 8.9787,E2 272.5318} C_DIS
LIN {X -134.8967,Y 2.8912,Z 171,A -179.4281,B 9.1365,C 0.2087,E1 8.9786,E2 270.7361} C_DIS
LIN {X -134.9252,Y -0.7608,Z 171,A -177.9188,B 9.1363,C 0.2138,E1 8.9786,E2 269.2333} C_DIS
LIN {X -134.8368,Y -4.921,Z 171,A -176.1249,B 9.1362,C 0.2185,E1 8.9787,E2 267.4378} C_DIS
LIN {X -134.6542,Y -8.5655,Z 171,A -174.5945,B 9.1361,C 0.2233,E1 8.979,E2 265.9111} C_DIS
LIN {X -134.3349,Y -12.6188,Z 171,A -172.8133,B 9.136,C 0.2274,E1 8.9794,E2 264.1247} C_DIS
LIN {X -133.9585,Y -16.1295,Z 171,A -171.3119,B 9.1359,C 0.2317,E1 8.9799,E2 262.6244} C_DIS
LIN {X -133.4097,Y -20.176,Z 171,A -169.4846,B 9.1358,C 0.2351,E1 8.9806,E2 260.7872} C_DIS
LIN {X -132.3628,Y -26.1841,Z 171,A -166.965,B 9.1356,C 0.2437,E1 8.9819,E2 258.2785} C_DIS
LIN {X -131.4919,Y -30.2473,Z 171,A -164.4603,B 9.1357,C 0.2363,E1 8.9835,E2 255.6837} C_DIS
LIN {X -130.2252,Y -35.3082,Z 171,A -162.9631,B 9.1353,C 0.2545,E1 8.9845,E2 254.2772} C_DIS
LIN {X -128.5292,Y -41.051,Z 171,A -160.6169,B 9.135,C 0.2647,E1 8.9863,E2 251.9571} C_DIS
LIN {X -127.4692,Y -44.233,Z 171,A -158.8445,B 9.135,C 0.2628,E1 8.9879,E2 250.143} C_DIS
LIN {X -126.3506,Y -47.3334,Z 171,A -157.4005,B 9.135,C 0.2659,E1 8.9893,E2 248.6946} C_DIS
LIN {X -125.0047,Y -50.7827,Z 171,A -155.8403,B 9.1348,C 0.2703,E1 8.9909,E2 247.137} C_DIS
LIN {X -123.642,Y -54.0169,Z 171,A -154.2486,B 9.1348,C 0.2725,E1 8.9927,E2 245.5338} C_DIS
LIN {X -121.0599,Y -59.5771,Z 171,A -151.9521,B 9.1344,C 0.2844,E1 8.9954,E2 243.2768} C_DIS
LIN {X -117.9671,Y -65.4922,Z 171,A -148.7293,B 9.1344,C 0.285,E1 8.9997,E2 240.0081} C_DIS
LIN {X -115.8221,Y -69.2151,Z 171,A -146.8626,B 9.1343,C 0.2888,E1 9.0023,E2 238.1372} C_DIS
LIN {X -113.4157,Y -73.0924,Z 171,A -144.6399,B 9.1343,C 0.2885,E1 9.0057,E2 235.8802} C_DIS
LIN {X -111.4968,Y -75.9868,Z 171,A -143.3893,B 9.134,C 0.2958,E1 9.0076,E2 234.6582} C_DIS
LIN {X -109.4756,Y -78.8713,Z 171,A -141.8492,B 9.134,C 0.2985,E1 9.0101,E2 233.1133} C_DIS
LIN {X -106.8617,Y -82.378,Z 171,A -139.9922,B 9.1338,C 0.3027,E1 9.0132,E2 231.2573} C_DIS
LIN {X -104.161,Y -85.7676,Z 171,A -138.0948,B 9.1338,C 0.3057,E1 9.0166,E2 229.3535} C_DIS
LIN {X -100.9759,Y -89.4949,Z 171,A -136.2697,B 9.1334,C 0.3146,E1 9.0199,E2 227.5612} C_DIS
LIN {X -98.1418,Y -92.5939,Z 171,A -134.4473,B 9.1333,C 0.3176,E1 9.0233,E2 225.7347} C_DIS
LIN {X -95.9426,Y -94.8713,Z 171,A -132.8252,B 9.1333,C 0.3155,E1 9.0266,E2 224.0785} C_DIS
LIN {X -93.5162,Y -97.2642,Z 171,A -131.2356,B 9.1333,C 0.3157,E1 9.0298,E2 222.4715} C_DIS
LIN {X -89.9627,Y -100.5593,Z 171,A -129.3137,B 9.1331,C 0.322,E1 9.0337,E2 220.5673} C_DIS
LIN {X -86.5037,Y -103.5502,Z 171,A -126.9444,B 9.1333,C 0.3178,E1 9.0389,E2 218.1449} C_DIS
LIN {X -83.0991,Y -106.3018,Z 171,A -125.5729,B 9.1329,C 0.3298,E1 9.0418,E2 216.8349} C_DIS
LIN {X -77.0844,Y -110.7404,Z 171,A -122.4279,B 9.1327,C 0.3355,E1 9.0489,E2 213.6943} C_DIS
LIN {X -73.9179,Y -112.8791,Z 171,A -120.6248,B 9.1327,C 0.3346,E1 9.0531,E2 211.8688} C_DIS
LIN {X -70.6199,Y -114.9708,Z 171,A -119.1377,B 9.1325,C 0.3402,E1 9.0566,E2 210.4032} C_DIS
LIN {X -67.6817,Y -116.7246,Z 171,A -117.5336,B 9.1325,C 0.3394,E1 9.0605,E2 208.7804} C_DIS
LIN {X -63.9273,Y -118.8224,Z 171,A -115.5764,B 9.1325,C 0.3394,E1 9.0653,E2 206.8068} C_DIS
LIN {X -58.2895,Y -121.6851,Z 171,A -113.3278,B 9.1321,C 0.3506,E1 9.0708,E2 204.6128} C_DIS
LIN {X -54.124,Y -123.5957,Z 171,A -110.9185,B 9.1323,C 0.3441,E1 9.0771,E2 202.1455} C_DIS
LIN {X -50.4245,Y -125.1491,Z 171,A -109.1963,B 9.1323,C 0.3454,E1 9.0815,E2 200.4208} C_DIS
LIN {X -46.3775,Y -126.7063,Z 171,A -107.442,B 9.1322,C 0.3488,E1 9.0861,E2 198.6773} C_DIS
LIN {X -39.3301,Y -129.0663,Z 171,A -104.3923,B 9.132,C 0.3533,E1 9.0942,E2 195.6406} C_DIS
LIN {X -36.3231,Y -129.9446,Z 171,A -103.0536,B 9.132,C 0.354,E1 9.0978,E2 194.3006} C_DIS
LIN {X -33.0007,Y -130.828,Z 171,A -101.5902,B 9.132,C 0.3548,E1 9.1017,E2 192.8365} C_DIS
LIN {X -30.0092,Y -131.5463,Z 171,A -100.2569,B 9.132,C 0.355,E1 9.1054,E2 191.4994} C_DIS
LIN {X -26.6814,Y -132.2616,Z 171,A -98.72,B 9.132,C 0.3539,E1 9.1096,E2 189.9506} C_DIS
LIN {X -22.2706,Y -133.0753,Z 171,A -96.8988,B 9.1319,C 0.3563,E1 9.1146,E2 188.1394} C_DIS
LIN {X -18.6216,Y -133.6356,Z 171,A -95.1766,B 9.1319,C 0.3537,E1 9.1194,E2 186.3972} C_DIS
LIN {X -13.9153,Y -134.2075,Z 171,A -93.3783,B 9.1319,C 0.3584,E1 9.1243,E2 184.6252} C_DIS
LIN {X -11.3514,Y -134.4477,Z 171,A -92.1705,B 9.1319,C 0.3563,E1 9.1277,E2 183.4026} C_DIS
LIN {X -6.7897,Y -134.7552,Z 171,A -90.1567,B 9.1319,C 0.3549,E1 9.1333,E2 181.3789} C_DIS
LIN {X 0.1805,Y -134.9272,Z 171,A -87.2528,B 9.1319,C 0.3559,E1 9.1414,E2 178.4809} C_DIS
LIN {X 0.1805,Y -134.9272,Z 171,A -87.2528,B 9.1319,C 0.3559,E1 9.1414,E2 178.4809} C_DIS
Enddeposition()
LIN {X 0.9824,Y -135.8322,Z 171,A -87.1078,B 9.0924,C 0.366,E1 9.1025,E2 178.4056} C_DIS
Startdeposition()
$VEL.CP = VEL_PRINT
LIN {X -5.2366,Y -135.7355,Z 171,A -89.9667,B 9.0922,C 0.371,E1 9.0945,E2 181.2957} C_DIS
LIN {X -10.8642,Y -135.4024,Z 171,A -92.6413,B 9.0919,C 0.3767,E1 9.0869,E2 184.0086} C_DIS
LIN {X -14.4488,Y -135.0657,Z 171,A -94.4565,B 9.0917,C 0.3822,E1 9.0818,E2 185.8613} C_DIS
LIN {X -18.118,Y -134.6234,Z 171,A -95.6753,B 9.092,C 0.3752,E1 9.0785,E2 187.0383} C_DIS
LIN {X -22.0003,Y -134.0433,Z 171,A -97.3479,B 9.092,C 0.375,E1 9.0739,E2 188.7135} C_DIS
LIN {X -25.3224,Y -133.4552,Z 171,A -98.7439,B 9.092,C 0.3739,E1 9.0701,E2 190.1066} C_DIS
LIN {X -28.7667,Y -132.7552,Z 171,A -100.256,B 9.092,C 0.3738,E1 9.0659,E2 191.6228} C_DIS
LIN {X -32.5585,Y -131.8786,Z 171,A -101.9654,B 9.092,C 0.3742,E1 9.0612,E2 193.3411} C_DIS
LIN {X -36.3744,Y -130.8755,Z 171,A -103.5522,B 9.0921,C 0.3716,E1 9.057,E2 194.9185} C_DIS
LIN {X -39.4843,Y -129.9712,Z 171,A -104.9493,B 9.0921,C 0.3712,E1 9.0532,E2 196.3198} C_DIS
LIN {X -44.0176,Y -128.5073,Z 171,A -107.0036,B 9.0921,C 0.3705,E1 9.0478,E2 198.38} C_DIS
LIN {X -47.5685,Y -127.2346,Z 171,A -108.5589,B 9.0923,C 0.3684,E1 9.0437,E2 199.9309} C_DIS
LIN {X -52.0463,Y -125.4699,Z 171,A -110.3749,B 9.0925,C 0.3624,E1 9.0391,E2 201.7203} C_DIS
LIN {X -55.0635,Y -124.1757,Z 171,A -112.0056,B 9.0924,C 0.3656,E1 9.0348,E2 203.3819} C_DIS
LIN {X -58.281,Y -122.698,Z 171,A -113.2829,B 9.0926,C 0.3599,E1 9.0316,E2 204.6323} C_DIS
LIN {X -61.0395,Y -121.3507,Z 171,A -114.7119,B 9.0926,C 0.3608,E1 9.028,E2 206.0781} C_DIS
LIN {X -64.4045,Y -119.5994,Z 171,A -116.4756,B 9.0926,C 0.3618,E1 9.0236,E2 207.8622} C_DIS
LIN {X -68.3201,Y -117.4069,Z 171,A -118.3935,B 9.0926,C 0.3598,E1 9.019,E2 209.7831} C_DIS
LIN {X -71.2969,Y -115.6233,Z 171,A -120.0558,B 9.0926,C 0.3613,E1 9.0149,E2 211.4699} C_DIS
LIN {X -74.0113,Y -113.9046,Z 171,A -121.2006,B 9.0928,C 0.3555,E1 9.0123,E2 212.5885} C_DIS
LIN {X -77.5476,Y -111.5271,Z 171,A -122.8702,B 9.093,C 0.3504,E1 9.0085,E2 214.2419} C_DIS
LIN {X -81.1347,Y -108.9454,Z 171,A -124.9024,B 9.093,C 0.3504,E1 9.0039,E2 216.2947} C_DIS
LIN {X -84.6848,Y -106.2094,Z 171,A -126.6589,B 9.0932,C 0.3448,E1 9,E2 218.0341} C_DIS
LIN {X -87.7732,Y -103.672,Z 171,A -128.5638,B 9.0932,C 0.3457,E1 8.9959,E2 219.9659} C_DIS
LIN {X -91.1602,Y -100.7064,Z 171,A -130.358,B 9.0934,C 0.3404,E1 8.9922,E2 221.7466} C_DIS
LIN {X -94.0867,Y -97.9782,Z 171,A -132.1613,B 9.0934,C 0.3392,E1 8.9885,E2 223.5637} C_DIS
LIN {X -97.2704,Y -94.8186,Z 171,A -134.1037,B 9.0935,C 0.3363,E1 8.9847,E2 225.5117} C_DIS
LIN {X -100.4388,Y -91.455,Z 171,A -136.0384,B 9.0937,C 0.332,E1 8.981,E2 227.4439} C_DIS
LIN {X -103.425,Y -88.0637,Z 171,A -137.9829,B 9.0937,C 0.3286,E1 8.9774,E2 229.3923} C_DIS
LIN {X -106.2882,Y -84.5858,Z 171,A -139.8705,B 9.0939,C 0.3243,E1 8.9741,E2 231.2776} C_DIS
LIN {X -108.414,Y -81.8434,Z 171,A -141.5887,B 9.0939,C 0.3253,E1 8.9712,E2 233.0265} C_DIS
LIN {X -110.3772,Y -79.176,Z 171,A -142.796,B 9.0941,C 0.3189,E1 8.9692,E2 234.2098} C_DIS
LIN {X -114.2311,Y -73.5071,Z 171,A -145.7628,B 9.0943,C 0.3134,E1 8.9646,E2 237.1844} C_DIS
LIN {X -116.6818,Y -69.5506,Z 171,A -147.7257,B 9.0945,C 0.3086,E1 8.9618,E2 239.1461} C_DIS
LIN {X -119.0204,Y -65.4693,Z 171,A -149.8669,B 9.0945,C 0.3063,E1 8.9588,E2 241.3055} C_DIS
LIN {X -121.0669,Y -61.5969,Z 171,A -151.4845,B 9.0948,C 0.2978,E1 8.9568,E2 242.8936} C_DIS
LIN {X -122.5371,Y -58.6179,Z 171,A -153.0467,B 9.0948,C 0.2968,E1 8.9548,E2 244.4748} C_DIS
LIN {X -124.4464,Y -54.4505,Z 171,A -154.9104,B 9.0951,C 0.2906,E1 8.9527,E2 246.3286} C_DIS
LIN {X -125.8157,Y -51.2056,Z 171,A -156.2916,B 9.0952,C 0.285,E1 8.9512,E2 247.6959} C_DIS
LIN {X -127.0923,Y -47.9486,Z 171,A -157.8819,B 9.0953,C 0.2829,E1 8.9496,E2 249.2993} C_DIS
LIN {X -128.2704,Y -44.701,Z 171,A -159.4808,B 9.0953,C 0.2813,E1 8.9481,E2 250.9145} C_DIS
LIN {X -129.2485,Y -41.7908,Z 171,A -160.7849,B 9.0955,C 0.2779,E1 8.947,E2 252.2188} C_DIS
LIN {X -131.5914,Y -33.6931,Z 171,A -164.5383,B 9.0957,C 0.2713,E1 8.9442,E2 255.9937} C_DIS
LIN {X -132.7266,Y -28.8992,Z 171,A -166.3065,B 9.096,C 0.2604,E1 8.9431,E2 257.7222} C_DIS
LIN {X -133.3418,Y -25.9154,Z 171,A -167.5778,B 9.096,C 0.2566,E1 8.9424,E2 258.9909} C_DIS
LIN {X -133.9989,Y -22.2662,Z 171,A -169.3079,B 9.0961,C 0.2548,E1 8.9415,E2 260.74} C_DIS
LIN {X -134.5823,Y -18.4319,Z 171,A -171.119,B 9.0961,C 0.253,E1 8.9408,E2 262.5712} C_DIS
LIN {X -135.027,Y -14.8082,Z 171,A -172.5774,B 9.0963,C 0.2473,E1 8.9403,E2 264.0182} C_DIS
LIN {X -135.3713,Y -11.2327,Z 171,A -174.1378,B 9.0964,C 0.2436,E1 8.9399,E2 265.5828} C_DIS
LIN {X -135.6518,Y -7.0839,Z 171,A -175.8928,B 9.0966,C 0.2386,E1 8.9396,E2 267.3363} C_DIS
LIN {X -135.8056,Y -2.9837,Z 171,A -177.7202,B 9.0966,C 0.2351,E1 8.9395,E2 269.1739} C_DIS
LIN {X -135.8372,Y 0.5181,Z 171,A -179.2298,B 9.0968,C 0.2314,E1 8.9395,E2 270.6861} C_DIS
LIN {X -135.746,Y 4.9677,Z 171,A 178.908,B 9.0968,C 0.2257,E1 8.9396,E2 272.5447} C_DIS
LIN {X -135.5732,Y 8.4519,Z 171,A 177.4428,B 9.097,C 0.2213,E1 8.9399,E2 274.0077} C_DIS
LIN {X -135.2609,Y 12.4991,Z 171,A 175.6809,B 9.0971,C 0.2171,E1 8.9403,E2 275.774} C_DIS
LIN {X -134.8742,Y 16.1389,Z 171,A 174.1345,B 9.0972,C 0.2127,E1 8.9408,E2 277.3191} C_DIS
LIN {X -134.2982,Y 20.387,Z 171,A 172.4937,B 9.0974,C 0.2048,E1 8.9414,E2 278.9378} C_DIS
LIN {X -133.765,Y 23.6325,Z 171,A 170.8757,B 9.0974,C 0.2045,E1 8.9422,E2 280.5825} C_DIS
LIN {X -133.0773,Y 27.2384,Z 171,A 169.3102,B 9.0974,C 0.2004,E1 8.943,E2 282.1485} C_DIS
LIN {X -132.2332,Y 31.0859,Z 171,A 167.5914,B 9.0976,C 0.1966,E1 8.9441,E2 283.8726} C_DIS
LIN {X -131.4641,Y 34.1929,Z 171,A 166.1548,B 9.0976,C 0.1942,E1 8.9451,E2 285.3184} C_DIS
LIN {X -130.4894,Y 37.7381,Z 171,A 164.6584,B 9.0977,C 0.1889,E1 8.9462,E2 286.8065} C_DIS
LIN {X -129.1892,Y 41.9766,Z 171,A 162.8078,B 9.0978,C 0.1834,E1 8.9477,E2 288.6529} C_DIS
LIN {X -126.2877,Y 50.0347,Z 171,A 158.9766,B 9.098,C 0.1771,E1 8.9515,E2 292.5069} C_DIS
LIN {X -124.7771,Y 53.6854,Z 171,A 157.4773,B 9.0981,C 0.1698,E1 8.9531,E2 293.9842} C_DIS
LIN {X -123.3494,Y 56.8888,Z 171,A 155.9735,B 9.0981,C 0.1663,E1 8.9548,E2 295.4894} C_DIS
LIN {X -122.0638,Y 59.5997,Z 171,A 154.6004,B 9.0981,C 0.1647,E1 8.9565,E2 296.8743} C_DIS
LIN {X -120.389,Y 62.9122,Z 171,A 152.746,B 9.0981,C 0.1654,E1 8.9589,E2 298.7618} C_DIS
LIN {X -118.722,Y 66.0081,Z 171,A 151.5161,B 9.0983,C 0.1574,E1 8.9605,E2 299.9597} C_DIS
LIN {X -116.6167,Y 69.6599,Z 171,A 149.6574,B 9.0983,C 0.1543,E1 8.9631,E2 301.8263} C_DIS
LIN {X -114.2921,Y 73.4118,Z 171,A 147.7895,B 9.0985,C 0.1498,E1 8.9659,E2 303.6931} C_DIS
LIN {X -111.9215,Y 76.9774,Z 171,A 146.1803,B 9.0985,C 0.1421,E1 8.9684,E2 305.2766} C_DIS
LIN {X -109.7206,Y 80.0843,Z 171,A 144.2713,B 9.0985,C 0.1433,E1 8.9716,E2 307.2206} C_DIS
LIN {X -106.974,Y 83.717,Z 171,A 142.3436,B 9.0986,C 0.1389,E1 8.9748,E2 309.1471} C_DIS
LIN {X -104.173,Y 87.1776,Z 171,A 140.6343,B 9.0987,C 0.1319,E1 8.9778,E2 310.8342} C_DIS
LIN {X -101.5608,Y 90.2077,Z 171,A 138.1276,B 9.0986,C 0.1418,E1 8.9826,E2 313.4373} C_DIS
LIN {X -97.8333,Y 94.2374,Z 171,A 136.3757,B 9.0988,C 0.1275,E1 8.9859,E2 315.1197} C_DIS
LIN {X -94.6617,Y 97.4225,Z 171,A 134.316,B 9.0988,C 0.1263,E1 8.99,E2 317.1972} C_DIS
LIN {X -91.3012,Y 100.5784,Z 171,A 132.0718,B 9.0988,C 0.1275,E1 8.9947,E2 319.4753} C_DIS
LIN {X -87.8521,Y 103.6049,Z 171,A 130.6237,B 9.0989,C 0.1156,E1 8.9977,E2 320.8633} C_DIS
LIN {X -84.6746,Y 106.2175,Z 171,A 128.8211,B 9.0989,C 0.1135,E1 9.0016,E2 322.6724} C_DIS
LIN {X -81.9143,Y 108.3605,Z 171,A 127.529,B 9.099,C 0.1077,E1 9.0044,E2 323.9412} C_DIS
LIN {X -76.7714,Y 112.0629,Z 171,A 124.6713,B 9.099,C 0.1064,E1 9.0109,E2 326.8188} C_DIS
LIN {X -73.3703,Y 114.3187,Z 171,A 122.9157,B 9.099,C 0.1042,E1 9.015,E2 328.577} C_DIS
LIN {X -69.7662,Y 116.5533,Z 171,A 121.2167,B 9.0991,C 0.0999,E1 9.0191,E2 330.2637} C_DIS
LIN {X -65.0836,Y 119.2311,Z 171,A 119.0187,B 9.0991,C 0.0952,E1 9.0244,E2 332.4504} C_DIS
LIN {X -57.5232,Y 123.056,Z 171,A 115.2631,B 9.0991,C 0.0937,E1 9.0338,E2 336.2251} C_DIS
LIN {X -54.3483,Y 124.4905,Z 171,A 113.7485,B 9.0992,C 0.0927,E1 9.0377,E2 337.744} C_DIS
LIN {X -51.4128,Y 125.7322,Z 171,A 112.3797,B 9.0992,C 0.0917,E1 9.0412,E2 339.1146} C_DIS
LIN {X -46.2217,Y 127.7302,Z 171,A 110.1106,B 9.0992,C 0.0878,E1 9.0471,E2 341.3727} C_DIS
LIN {X -43.3076,Y 128.748,Z 171,A 108.7381,B 9.0992,C 0.0878,E1 9.0508,E2 342.7528} C_DIS
LIN {X -39.9149,Y 129.8394,Z 171,A 107.3129,B 9.0992,C 0.0851,E1 9.0545,E2 344.1674} C_DIS
LIN {X -37.3886,Y 130.5917,Z 171,A 105.8099,B 9.0992,C 0.0913,E1 9.0587,E2 345.7166} C_DIS
LIN {X -34.0486,Y 131.5012,Z 171,A 104.5813,B 9.0992,C 0.0859,E1 9.0619,E2 346.9165} C_DIS
LIN {X -30.3067,Y 132.4121,Z 171,A 103.1038,B 9.0993,C 0.0821,E1 9.0659,E2 348.3753} C_DIS
LIN {X -26.8819,Y 133.1498,Z 171,A 101.5581,B 9.0993,C 0.0824,E1 9.0701,E2 349.9282} C_DIS
LIN {X -22.7038,Y 133.9259,Z 171,A 99.7456,B 9.0993,C 0.0819,E1 9.0751,E2 351.742} C_DIS
LIN {X -19.1749,Y 134.4761,Z 171,A 98.2593,B 9.0993,C 0.0808,E1 9.0792,E2 353.225} C_DIS
LIN {X -15.2449,Y 134.98,Z 171,A 96.4951,B 9.0993,C 0.0819,E1 9.0841,E2 354.9995} C_DIS
LIN {X -11.5956,Y 135.3406,Z 171,A 95.0056,B 9.0993,C 0.0804,E1 9.0883,E2 356.4813} C_DIS
LIN {X -7.7651,Y 135.6156,Z 171,A 93.3083,B 9.0993,C 0.0815,E1 9.093,E2 358.1871} C_DIS
LIN {X -3.6739,Y 135.7868,Z 171,A 91.6553,B 9.0993,C 0.0799,E1 9.0976,E2 359.8303} C_DIS
LIN {X 0.4788,Y 135.8359,Z 171,A 89.912,B 9.0993,C 0.0797,E1 9.1025,E2 361.5718} C_DIS
LIN {X 4.0872,Y 135.7753,Z 171,A 88.2839,B 9.0993,C 0.0818,E1 9.107,E2 363.212} C_DIS
LIN {X 8.3266,Y 135.581,Z 171,A 86.6334,B 9.0993,C 0.0793,E1 9.1116,E2 364.845} C_DIS
LIN {X 11.8583,Y 135.3184,Z 171,A 85.1097,B 9.0993,C 0.0802,E1 9.1159,E2 366.3717} C_DIS
LIN {X 15.8923,Y 134.9036,Z 171,A 83.4485,B 9.0993,C 0.0798,E1 9.1204,E2 368.0263} C_DIS
LIN {X 19.4314,Y 134.4394,Z 171,A 81.8925,B 9.0993,C 0.0813,E1 9.1248,E2 369.5879} C_DIS
LIN {X 23.6422,Y 133.7633,Z 171,A 80.1496,B 9.0993,C 0.081,E1 9.1295,E2 371.3235} C_DIS
LIN {X 26.8865,Y 133.1489,Z 171,A 78.708,B 9.0993,C 0.0827,E1 9.1335,E2 372.7706} C_DIS
LIN {X 30.135,Y 132.4513,Z 171,A 77.2906,B 9.0993,C 0.0839,E1 9.1374,E2 374.1896} C_DIS
LIN {X 33.8889,Y 131.5418,Z 171,A 75.7084,B 9.0993,C 0.0841,E1 9.1417,E2 375.7658} C_DIS
LIN {X 37.7246,Y 130.4933,Z 171,A 73.8145,B 9.0993,C 0.0897,E1 9.1468,E2 377.6855} C_DIS
LIN {X 42.5839,Y 128.989,Z 171,A 71.9197,B 9.0993,C 0.0865,E1 9.1518,E2 379.5497} C_DIS
LIN {X 46.1975,Y 127.7389,Z 171,A 70.2463,B 9.0993,C 0.0892,E1 9.1562,E2 381.2302} C_DIS
LIN {X 49.9394,Y 126.3246,Z 171,A 68.3338,B 9.0992,C 0.0955,E1 9.1613,E2 383.1698} C_DIS
LIN {X 53.0363,Y 125.0564,Z 171,A 67.1053,B 9.0992,C 0.0933,E1 9.1644,E2 384.3761} C_DIS
LIN {X 56.7758,Y 123.4017,Z 171,A 65.4897,B 9.0992,C 0.0931,E1 9.1684,E2 385.9784} C_DIS
LIN {X 59.8476,Y 121.9415,Z 171,A 64.1878,B 9.0992,C 0.0922,E1 9.1717,E2 387.2642} C_DIS
LIN {X 62.8495,Y 120.4219,Z 171,A 62.7072,B 9.0992,C 0.0953,E1 9.1754,E2 388.7523} C_DIS
LIN {X 66.3503,Y 118.5311,Z 171,A 61.0046,B 9.0992,C 0.0981,E1 9.1795,E2 390.4581} C_DIS
LIN {X 70.9029,Y 115.8652,Z 171,A 58.7168,B 9.0991,C 0.1026,E1 9.1851,E2 392.7536} C_DIS
LIN {X 74.5892,Y 113.5271,Z 171,A 57.1255,B 9.0991,C 0.1003,E1 9.1887,E2 394.3148} C_DIS
LIN {X 77.5428,Y 111.5305,Z 171,A 55.4071,B 9.0991,C 0.1072,E1 9.1927,E2 396.0595} C_DIS
LIN {X 81.1859,Y 108.9072,Z 171,A 53.5398,B 9.0991,C 0.1098,E1 9.1969,E2 397.924} C_DIS
LIN {X 84.2042,Y 106.5914,Z 171,A 51.9339,B 9.099,C 0.1127,E1 9.2005,E2 399.5303} C_DIS
LIN {X 87.6405,Y 103.7847,Z 171,A 50.2539,B 9.099,C 0.112,E1 9.204,E2 401.1875} C_DIS
LIN {X 89.9609,Y 101.779,Z 171,A 48.8559,B 9.099,C 0.1167,E1 9.207,E2 402.5986} C_DIS
LIN {X 92.9232,Y 99.0826,Z 171,A 47.0938,B 9.0989,C 0.1215,E1 9.2106,E2 404.37} C_DIS
LIN {X 96.0878,Y 96.0167,Z 171,A 45.264,B 9.0989,C 0.1246,E1 9.2143,E2 406.1969} C_DIS
LIN {X 99.1348,Y 92.8676,Z 171,A 43.4286,B 9.0988,C 0.1282,E1 9.2178,E2 408.0314} C_DIS
LIN {X 102.2018,Y 89.4806,Z 171,A 41.57,B 9.0988,C 0.1309,E1 9.2213,E2 409.8824} C_DIS
LIN {X 104.9872,Y 86.1958,Z 171,A 40.0668,B 9.0988,C 0.128,E1 9.2239,E2 411.348} C_DIS
LIN {X 107.2091,Y 83.4159,Z 171,A 38.2759,B 9.0986,C 0.1377,E1 9.2271,E2 413.175} C_DIS
LIN {X 109.8859,Y 79.8564,Z 171,A 36.4468,B 9.0986,C 0.141,E1 9.2301,E2 414.9991} C_DIS
LIN {X 112.4938,Y 76.1385,Z 171,A 34.5613,B 9.0986,C 0.1449,E1 9.2331,E2 416.8819} C_DIS
LIN {X 114.932,Y 72.4056,Z 171,A 32.721,B 9.0985,C 0.1485,E1 9.2358,E2 418.7182} C_DIS
LIN {X 117.2723,Y 68.5508,Z 171,A 30.304,B 9.0982,C 0.1645,E1 9.2394,E2 421.199} C_DIS
LIN {X 119.6856,Y 64.244,Z 171,A 28.6775,B 9.0982,C 0.1598,E1 9.2415,E2 422.7713} C_DIS
LIN {X 121.5499,Y 60.6414,Z 171,A 27.0945,B 9.0982,C 0.1614,E1 9.2434,E2 424.3397} C_DIS
LIN {X 123.2321,Y 57.1424,Z 171,A 25.5535,B 9.0982,C 0.1635,E1 9.2453,E2 425.8698} C_DIS
LIN {X 124.5538,Y 54.202,Z 171,A 24.3175,B 9.0982,C 0.1643,E1 9.2466,E2 427.0915} C_DIS
LIN {X 125.8302,Y 51.1696,Z 171,A 23.0058,B 9.0982,C 0.1663,E1 9.248,E2 428.3948} C_DIS
LIN {X 127.035,Y 48.1016,Z 171,A 21.4648,B 9.098,C 0.1734,E1 9.2496,E2 429.9554} C_DIS
LIN {X 128.4316,Y 44.2358,Z 171,A 19.7218,B 9.098,C 0.1783,E1 9.2512,E2 431.7008} C_DIS
LIN {X 129.6419,Y 40.559,Z 171,A 17.8628,B 9.0978,C 0.1879,E1 9.2528,E2 433.5888} C_DIS
LIN {X 130.5953,Y 37.3761,Z 171,A 16.6664,B 9.0978,C 0.1872,E1 9.2538,E2 434.7612} C_DIS
LIN {X 131.5993,Y 33.6621,Z 171,A 15.1761,B 9.0978,C 0.1887,E1 9.2548,E2 436.2363} C_DIS
LIN {X 132.4006,Y 30.357,Z 171,A 13.7315,B 9.0976,C 0.193,E1 9.2557,E2 437.6833} C_DIS
LIN {X 133.2011,Y 26.6299,Z 171,A 12.0737,B 9.0976,C 0.1987,E1 9.2567,E2 439.3486} C_DIS
LIN {X 133.963,Y 22.4814,Z 171,A 10.3988,B 9.0975,C 0.2014,E1 9.2575,E2 441.0122} C_DIS
LIN {X 134.5885,Y 18.3838,Z 171,A 8.6832,B 9.0974,C 0.2057,E1 9.2582,E2 442.7253} C_DIS
LIN {X 135.0248,Y 14.8293,Z 171,A 7.2037,B 9.0973,C 0.2093,E1 9.2586,E2 444.2023} C_DIS
LIN {X 135.3594,Y 11.374,Z 171,A 5.7519,B 9.0972,C 0.2133,E1 9.259,E2 445.6538} C_DIS
LIN {X 135.6441,Y 7.2375,Z 171,A 4.0182,B 9.0971,C 0.218,E1 9.2593,E2 447.3872} C_DIS
LIN {X 135.7901,Y 3.5535,Z 171,A 2.4541,B 9.097,C 0.2227,E1 9.2594,E2 448.9539} C_DIS
LIN {X 135.8374,Y -0.4895,Z 171,A 0.7538,B 9.0969,C 0.2276,E1 9.2594,E2 450.6552} C_DIS
LIN {X 135.7793,Y -3.9427,Z 171,A -0.5595,B 9.0969,C 0.2285,E1 9.2594,E2 451.952} C_DIS
LIN {X 135.6435,Y -7.2501,Z 171,A -2.077,B 9.0967,C 0.2353,E1 9.2592,E2 453.4859} C_DIS
LIN {X 135.3338,Y -11.6767,Z 171,A -3.7952,B 9.0967,C 0.2373,E1 9.2588,E2 455.1869} C_DIS
LIN {X 134.9182,Y -15.77,Z 171,A -5.5141,B 9.0965,C 0.242,E1 9.2583,E2 456.9054} C_DIS
LIN {X 134.5026,Y -18.9894,Z 171,A -6.9096,B 9.0964,C 0.2465,E1 9.2578,E2 458.3055} C_DIS
LIN {X 133.8841,Y -22.9541,Z 171,A -8.5282,B 9.0963,C 0.2497,E1 9.257,E2 459.9167} C_DIS
LIN {X 133.1326,Y -26.9668,Z 171,A -10.2059,B 9.0962,C 0.2536,E1 9.2562,E2 461.5906} C_DIS
LIN {X 132.472,Y -30.0445,Z 171,A -11.5607,B 9.096,C 0.258,E1 9.2553,E2 462.9501} C_DIS
LIN {X 131.7524,Y -33.0589,Z 171,A -12.9961,B 9.0959,C 0.2647,E1 9.2544,E2 464.4028} C_DIS
LIN {X 130.5044,Y -37.6866,Z 171,A -14.8088,B 9.0959,C 0.2657,E1 9.253,E2 466.1916} C_DIS
LIN {X 129.4594,Y -41.1307,Z 171,A -16.0883,B 9.0959,C 0.2645,E1 9.252,E2 467.4428} C_DIS
LIN {X 128.5151,Y -43.995,Z 171,A -17.6048,B 9.0956,C 0.2736,E1 9.2506,E2 468.9912} C_DIS
LIN {X 127.4671,Y -46.948,Z 171,A -18.9631,B 9.0955,C 0.2781,E1 9.2493,E2 470.3555} C_DIS
LIN {X 126.0936,Y -50.5162,Z 171,A -20.4336,B 9.0955,C 0.2793,E1 9.2478,E2 471.81} C_DIS
LIN {X 124.7771,Y -53.6854,Z 171,A -21.7556,B 9.0954,C 0.2804,E1 9.2464,E2 473.1177} C_DIS
LIN {X 122.9153,Y -57.8252,Z 171,A -23.7859,B 9.0951,C 0.2881,E1 9.244,E2 475.1646} C_DIS
LIN {X 121.3474,Y -61.046,Z 171,A -25.2499,B 9.0951,C 0.2911,E1 9.2422,E2 476.6244} C_DIS
LIN {X 119.4625,Y -64.6591,Z 171,A -27.052,B 9.0949,C 0.2974,E1 9.2399,E2 478.4387} C_DIS
LIN {X 118.0216,Y -67.2521,Z 171,A -28.3646,B 9.0947,C 0.302,E1 9.238,E2 479.7602} C_DIS
LIN {X 115.4529,Y -71.5724,Z 171,A -30.3339,B 9.0947,C 0.304,E1 9.2352,E2 481.7129} C_DIS
LIN {X 113.093,Y -75.246,Z 171,A -32.1739,B 9.0945,C 0.3086,E1 9.2324,E2 483.5546} C_DIS
Enddeposition()
END
